KUKA KRL program: EPS_2_25694_BP01_A_20251117072354.src

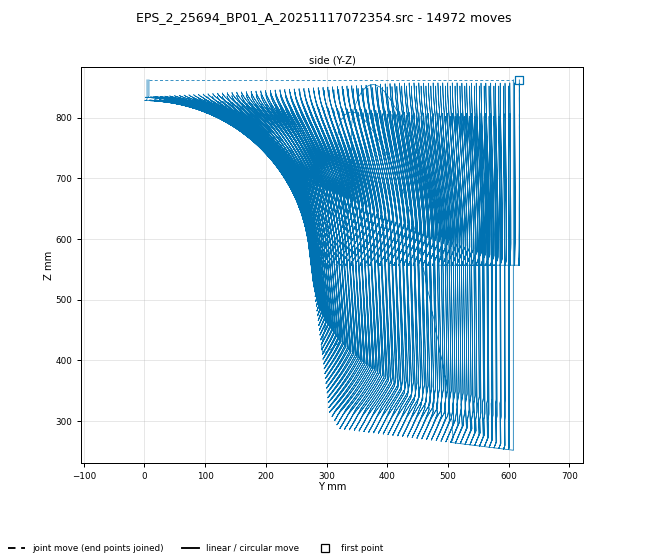
[picture p0: tool path of EPS_2_25694_BP01_A_20251117072354.src, 14972 of 14974 moves have a stored position in this frame; points joined in program order, loops and branches not executed]
&ACCESS RVP
&REL 4
&COMMENT QRS 19112012
&PARAM EDITMASK = *
DEF PART()
EXT BAS (BAS_COMMAND :IN,REAL :IN )
INT I
BAS (#INITMOV,0 )

;KUKA QRS Post kuka4.cps  Date:22-06-2017 !

File_ID=2910

QRS_PRE_INIT()

;Init var - Until changes are made in qrs_pre_init
Outlet_Square_prg=0
Inlet_1_Square_prg=0
Inlet_2_Square_prg=0
Inlet_3_Square_prg=0
Inlet_4_Square_prg=0
Inlet_5_Square_prg=0

Outlet_1={X 0.000, Y 425.000, Z 586.000, B 0.000, E1 0.000 }
Inlet_1={X 0.000, Y 466.000, Z 574.000, B 0.000, E1 180.000 }
Outlet_1_type=533
Inlet_1_type=457
;QRS#1=Sidecore dimensions
;QRS#2=525-21" Concrete
;QRS#3=450-18" Concrete
;QRS#4=
;QRS#5=
;QRS#6=
;QRS#7=
;QRS#8=
;QRS#9=S306-32
;QRS#10=28A PSX-2
;QRS#11=
;QRS#12=
;QRS#13=
;QRS#14=
;QRS#15=
;QRS#16=1220x127x1219 4'
;QRS#17=EPS Height
;QRS#18=852,5
;QRS#19=*
;QRS#20= UPDATED VERSION 22-06-2017
;QRS#21=*
Outlet_Square=0250
Inlet_1_Square=0250
Inlet_2_Square=0
Inlet_3_Square=0
Inlet_4_Square=0
Inlet_5_Square=0
Mill_Square=1
Outlet_Square_Prg=263
Inlet_1_Square_prg=274

QRS_INIT()

$ADVANCE=5

; T1
PTP {E1 171.043,E2 171.043}
PTP {X 0,Y 617.776,A -85,B 0,C 180,E1 171.043,E2 171.043,E3 0,E4 0,E5 0,E6 0}
QRS_SPEED_INIT()
LIN {X 0,Y 617.776,Z 862.5,A -85,B 0,C 180,E1 171.043,E2 171.043,E3 0,E4 0,E5 0,E6 0} C_VEL
LIN {X 0,Y 617.776,Z 559.03,A -85,B 0,C 180,E1 171.043,E2 171.043} C_VEL
LIN {X 0,Y 617.813,Z 557.03,A -85,B 0,C 180,E1 171.228,E2 171.228} C_VEL
LIN {X 0,Y 617.994,Z 557.03,A -85,B 0,C 180,E1 171.886,E2 171.886} C_VEL
LIN {X 0,Y 618.06,Z 557.03,A -85,B 0,C 180,E1 176.532,E2 176.532} C_VEL
LIN {X 0,Y 618.033,Z 557.03,A -85,B 0,C 180,E1 181.155,E2 181.155} C_VEL
LIN {X 0,Y 617.978,Z 557.03,A -85,B 0,C 180,E1 185.787,E2 185.787} C_VEL
LIN {X 0,Y 617.994,Z 557.03,A -85,B 0,C 180,E1 190.456,E2 190.456} C_VEL
LIN {X 0,Y 617.919,Z 557.03,A -85,B 0,C 180,E1 195.199,E2 195.199} C_VEL
LIN {X 0,Y 617.921,Z 557.03,A -85,B 0,C 180,E1 200.05,E2 200.05} C_VEL
LIN {X 0,Y 617.439,Z 557.03,A -85,B 0,C 180,E1 202.548,E2 202.548} C_VEL
LIN {X 0,Y 617.89,Z 557.03,A -85,B 0,C 180,E1 205.057,E2 205.057} C_VEL
LIN {X 0,Y 617.413,Z 557.03,A -85,B 0,C 180,E1 207.659,E2 207.659} C_VEL
LIN {X 0,Y 617.896,Z 557.03,A -85,B 0,C 180,E1 210.277,E2 210.277} C_VEL
LIN {X 0,Y 617.343,Z 557.03,A -85,B 0,C 180,E1 213.025,E2 213.025} C_VEL
LIN {X 0,Y 617.808,Z 557.03,A -85,B 0,C 180,E1 215.799,E2 215.799} C_VEL
LIN {X 0,Y 617.581,Z 557.03,A -85,B 0,C 180,E1 218.103,E2 218.103} C_VEL
LIN {X 0,Y 617.561,Z 557.03,A -85,B 0,C 180,E1 218.721,E2 218.721} C_VEL
LIN {X 0,Y 617.791,Z 557.03,A -85,B 0,C 180,E1 221.731,E2 221.731} C_VEL
LIN {X 0,Y 617.868,Z 557.03,A -85,B 0,C 180,E1 225.1,E2 225.1} C_VEL
LIN {X 0,Y 617.445,Z 557.03,A -85,B 0,C 180,E1 228.309,E2 228.309} C_VEL
LIN {X 0,Y 617.791,Z 557.03,A -85,B 0,C 180,E1 231.298,E2 231.298} C_VEL
LIN {X 0,Y 617.736,Z 557.03,A -85,B 0,C 180,E1 235.8,E2 235.8} C_VEL
LIN {X 0,Y 617.923,Z 557.03,A -85,B 0,C 180,E1 237.011,E2 237.011} C_VEL
LIN {X 0,Y 618.028,Z 557.03,A -85,B 0,C 180,E1 240.51,E2 240.51} C_VEL
LIN {X 0,Y 617.97,Z 557.03,A -85,B 0,C 180,E1 240.75,E2 240.75} C_VEL
LIN {X 0,Y 616.889,Z 557.03,A -85,B 0,C 180,E1 240.936,E2 240.936} C_VEL
LIN {X 0,Y 616.577,Z 557.502,A -85,B 0,C 180,E1 240.975,E2 240.975} C_VEL
LIN {X 0,Y 617.559,Z 570.177,A -85,B 0,C 180,E1 241.191,E2 241.191} C_VEL
LIN {X 0,Y 617.762,Z 600.266,A -85,B 0,C 180,E1 241.598,E2 241.598} C_VEL
LIN {X 0,Y 617.686,Z 612.976,A -85,B 0,C 180,E1 241.802,E2 241.802} C_VEL
LIN {X 0,Y 617.749,Z 625.832,A -85,B 0,C 180,E1 242.076,E2 242.076} C_VEL
LIN {X 0,Y 617.694,Z 639.689,A -85,B 0,C 180,E1 242.437,E2 242.437} C_VEL
LIN {X 0,Y 617.798,Z 652.671,A -85,B 0,C 180,E1 242.849,E2 242.849} C_VEL
LIN {X 0,Y 617.803,Z 663.961,A -85,B 0,C 180,E1 243.254,E2 243.254} C_VEL
LIN {X 0,Y 617.861,Z 675.827,A -85,B 0,C 180,E1 243.741,E2 243.741} C_VEL
LIN {X 0,Y 617.923,Z 689.601,A -85,B 0,C 180,E1 244.386,E2 244.386} C_VEL
LIN {X 0,Y 617.876,Z 701.688,A -85,B 0,C 180,E1 245.016,E2 245.016} C_VEL
LIN {X 0,Y 617.897,Z 713.952,A -85,B 0,C 180,E1 245.732,E2 245.732} C_VEL
LIN {X 0,Y 617.922,Z 724.145,A -85,B 0,C 180,E1 246.381,E2 246.381} C_VEL
LIN {X 0,Y 617.934,Z 735.43,A -85,B 0,C 180,E1 247.172,E2 247.172} C_VEL
LIN {X 0,Y 617.917,Z 745.514,A -85,B 0,C 180,E1 247.939,E2 247.939} C_VEL
LIN {X 0,Y 617.886,Z 756.654,A -85,B 0,C 180,E1 248.87,E2 248.87} C_VEL
LIN {X 0,Y 617.923,Z 766.773,A -85,B 0,C 180,E1 249.797,E2 249.797} C_VEL
LIN {X 0,Y 617.933,Z 775.518,A -85,B 0,C 180,E1 250.667,E2 250.667} C_VEL
LIN {X 0,Y 617.881,Z 782.638,A -85,B 0,C 180,E1 251.422,E2 251.422} C_VEL
LIN {X 0,Y 617.901,Z 791.021,A -85,B 0,C 180,E1 252.392,E2 252.392} C_VEL
LIN {X 0,Y 617.982,Z 799.193,A -85,B 0,C 180,E1 253.428,E2 253.428} C_VEL
LIN {X 0,Y 617.836,Z 807.711,A -85,B 0,C 180,E1 254.61,E2 254.61} C_VEL
LIN {X 0,Y 617.888,Z 814.772,A -85,B 0,C 180,E1 255.697,E2 255.697} C_VEL
LIN {X 0,Y 617.959,Z 820.124,A -85,B 0,C 180,E1 256.591,E2 256.591} C_VEL
LIN {X 0,Y 617.783,Z 826.565,A -85,B 0,C 180,E1 257.773,E2 257.773} C_VEL
LIN {X 0,Y 617.807,Z 832.247,A -85,B 0,C 180,E1 258.953,E2 258.953} C_VEL
LIN {X 0,Y 617.977,Z 836.456,A -85,B 0,C 180,E1 259.949,E2 259.949} C_VEL
LIN {X 0,Y 617.803,Z 841.446,A -85,B 0,C 180,E1 261.247,E2 261.247} C_VEL
LIN {X 0,Y 617.803,Z 845.018,A -85,B 0,C 180,E1 262.35,E2 262.35} C_VEL
LIN {X 0,Y 617.953,Z 848.842,A -85,B 0,C 180,E1 263.749,E2 263.749} C_VEL
LIN {X 0,Y 617.736,Z 851.904,A -85,B 0,C 180,E1 265.14,E2 265.14} C_VEL
LIN {X 0,Y 617.832,Z 854.096,A -85,B 0,C 180,E1 266.531,E2 266.531} C_VEL
LIN {X 0,Y 617.988,Z 855.163,A -85,B 0,C 180,E1 267.458,E2 267.458} C_VEL
LIN {X 0,Y 617.747,Z 856.216,A -85,B 0,C 180,E1 268.844,E2 268.844} C_VEL
LIN {X 0,Y 617.992,Z 856.149,A -85,B 0,C 180,E1 271.155,E2 271.155} C_VEL
LIN {X 0,Y 617.755,Z 855.226,A -85,B 0,C 180,E1 272.543,E2 272.543} C_VEL
LIN {X 0,Y 617.755,Z 854.116,A -85,B 0,C 180,E1 273.469,E2 273.469} C_VEL
LIN {X 0,Y 617.985,Z 851.839,A -85,B 0,C 180,E1 274.858,E2 274.858} C_VEL
LIN {X 0,Y 617.799,Z 848.881,A -85,B 0,C 180,E1 276.253,E2 276.253} C_VEL
LIN {X 0,Y 617.848,Z 845.007,A -85,B 0,C 180,E1 277.649,E2 277.649} C_VEL
LIN {X 0,Y 617.932,Z 841.117,A -85,B 0,C 180,E1 278.831,E2 278.831} C_VEL
LIN {X 0,Y 617.775,Z 836.414,A -85,B 0,C 180,E1 280.075,E2 280.075} C_VEL
LIN {X 0,Y 617.825,Z 832.243,A -85,B 0,C 180,E1 281.047,E2 281.047} C_VEL
LIN {X 0,Y 617.969,Z 826.527,A -85,B 0,C 180,E1 282.224,E2 282.224} C_VEL
LIN {X 0,Y 617.83,Z 820.149,A -85,B 0,C 180,E1 283.411,E2 283.411} C_VEL
LIN {X 0,Y 617.902,Z 811.935,A -85,B 0,C 180,E1 284.75,E2 284.75} C_VEL
LIN {X 0,Y 617.938,Z 805.132,A -85,B 0,C 180,E1 285.758,E2 285.758} C_VEL
LIN {X 0,Y 617.865,Z 798.318,A -85,B 0,C 180,E1 286.693,E2 286.693} C_VEL
LIN {X 0,Y 617.91,Z 789.904,A -85,B 0,C 180,E1 287.74,E2 287.74} C_VEL
LIN {X 0,Y 617.968,Z 781.813,A -85,B 0,C 180,E1 288.665,E2 288.665} C_VEL
LIN {X 0,Y 617.898,Z 771.905,A -85,B 0,C 180,E1 289.703,E2 289.703} C_VEL
LIN {X 0,Y 617.915,Z 763.533,A -85,B 0,C 180,E1 290.511,E2 290.511} C_VEL
LIN {X 0,Y 617.932,Z 753.036,A -85,B 0,C 180,E1 291.438,E2 291.438} C_VEL
LIN {X 0,Y 617.906,Z 743.499,A -85,B 0,C 180,E1 292.217,E2 292.217} C_VEL
LIN {X 0,Y 617.904,Z 733.654,A -85,B 0,C 180,E1 292.959,E2 292.959} C_VEL
LIN {X 0,Y 617.855,Z 722.087,A -85,B 0,C 180,E1 293.756,E2 293.756} C_VEL
LIN {X 0,Y 617.9,Z 709.883,A -85,B 0,C 180,E1 294.513,E2 294.513} C_VEL
LIN {X 0,Y 617.869,Z 698.891,A -85,B 0,C 180,E1 295.137,E2 295.137} C_VEL
LIN {X 0,Y 617.811,Z 688.028,A -85,B 0,C 180,E1 295.699,E2 295.699} C_VEL
LIN {X 0,Y 617.891,Z 673.877,A -85,B 0,C 180,E1 296.338,E2 296.338} C_VEL
LIN {X 0,Y 617.852,Z 660.675,A -85,B 0,C 180,E1 296.865,E2 296.865} C_VEL
LIN {X 0,Y 617.731,Z 650.373,A -85,B 0,C 180,E1 297.236,E2 297.236} C_VEL
LIN {X 0,Y 617.857,Z 634.521,A -85,B 0,C 180,E1 297.699,E2 297.699} C_VEL
LIN {X 0,Y 617.754,Z 621.706,A -85,B 0,C 180,E1 298.018,E2 298.018} C_VEL
LIN {X 0,Y 617.687,Z 613.02,A -85,B 0,C 180,E1 298.197,E2 298.197} C_VEL
LIN {X 0,Y 617.736,Z 606.549,A -85,B 0,C 180,E1 298.307,E2 298.307} C_VEL
LIN {X 0,Y 617.744,Z 594.08,A -85,B 0,C 180,E1 298.49,E2 298.49} C_VEL
LIN {X 0,Y 617.654,Z 580.796,A -85,B 0,C 180,E1 298.667,E2 298.667} C_VEL
LIN {X 0,Y 617.292,Z 566.02,A -85,B 0,C 180,E1 298.877,E2 298.877} C_VEL
LIN {X 0,Y 616.884,Z 557.03,A -85,B 0,C 180,E1 299.063,E2 299.063} C_VEL
LIN {X 0,Y 617.909,Z 557.03,A -85,B 0,C 180,E1 299.23,E2 299.23} C_VEL
LIN {X 0,Y 618.035,Z 557.03,A -85,B 0,C 180,E1 299.444,E2 299.444} C_VEL
LIN {X 0,Y 617.919,Z 557.03,A -85,B 0,C 180,E1 302.989,E2 302.989} C_VEL
LIN {X 0,Y 617.722,Z 557.03,A -85,B 0,C 180,E1 304.198,E2 304.198} C_VEL
LIN {X 0,Y 617.789,Z 557.03,A -85,B 0,C 180,E1 308.703,E2 308.703} C_VEL
LIN {X 0,Y 617.443,Z 557.03,A -85,B 0,C 180,E1 311.758,E2 311.758} C_VEL
LIN {X 0,Y 617.868,Z 557.03,A -85,B 0,C 180,E1 314.9,E2 314.9} C_VEL
LIN {X 0,Y 617.791,Z 557.03,A -85,B 0,C 180,E1 318.271,E2 318.271} C_VEL
LIN {X 0,Y 617.554,Z 557.03,A -85,B 0,C 180,E1 321.278,E2 321.278} C_VEL
LIN {X 0,Y 617.58,Z 557.03,A -85,B 0,C 180,E1 321.897,E2 321.897} C_VEL
LIN {X 0,Y 617.801,Z 557.03,A -85,B 0,C 180,E1 324.201,E2 324.201} C_VEL
LIN {X 0,Y 617.345,Z 557.03,A -85,B 0,C 180,E1 326.975,E2 326.975} C_VEL
LIN {X 0,Y 617.887,Z 557.03,A -85,B 0,C 180,E1 329.722,E2 329.722} C_VEL
LIN {X 0,Y 617.405,Z 557.03,A -85,B 0,C 180,E1 332.34,E2 332.34} C_VEL
LIN {X 0,Y 617.882,Z 557.03,A -85,B 0,C 180,E1 334.943,E2 334.943} C_VEL
LIN {X 0,Y 617.431,Z 557.03,A -85,B 0,C 180,E1 337.451,E2 337.451} C_VEL
LIN {X 0,Y 617.935,Z 557.03,A -85,B 0,C 180,E1 339.951,E2 339.951} C_VEL
LIN {X 0,Y 618,Z 557.03,A -85,B 0,C 180,E1 343.636,E2 343.636} C_VEL
LIN {X 0,Y 617.991,Z 557.03,A -85,B 0,C 180,E1 349.544,E2 349.544} C_VEL
LIN {X 0,Y 617.989,Z 557.03,A -85,B 0,C 180,E1 354.213,E2 354.213} C_VEL
LIN {X 0,Y 618.039,Z 557.03,A -85,B 0,C 180,E1 358.845,E2 358.845} C_VEL
LIN {X 0,Y 618.057,Z 557.03,A -85,B 0,C 180,E1 363.468,E2 363.468} C_VEL
LIN {X 0,Y 618.001,Z 557.03,A -85,B 0,C 180,E1 368.114,E2 368.114} C_VEL
LIN {X 0,Y 617.989,Z 557.03,A -85,B 0,C 180,E1 372.815,E2 372.815} C_VEL
LIN {X 0,Y 617.976,Z 557.03,A -85,B 0,C 180,E1 377.606,E2 377.606} C_VEL
LIN {X 0,Y 617.778,Z 557.03,A -85,B 0,C 180,E1 378.555,E2 378.555} C_VEL
LIN {X 0,Y 617.925,Z 557.03,A -85,B 0,C 180,E1 382.53,E2 382.53} C_VEL
LIN {X 0,Y 617.433,Z 557.03,A -85,B 0,C 180,E1 385.077,E2 385.077} C_VEL
LIN {X 0,Y 617.885,Z 557.03,A -85,B 0,C 180,E1 387.636,E2 387.636} C_VEL
LIN {X 0,Y 617.381,Z 557.03,A -85,B 0,C 180,E1 390.305,E2 390.305} C_VEL
LIN {X 0,Y 617.86,Z 557.03,A -85,B 0,C 180,E1 392.994,E2 392.994} C_VEL
LIN {X 0,Y 617.716,Z 557.03,A -85,B 0,C 180,E1 394.2,E2 394.2} C_VEL
LIN {X 0,Y 617.789,Z 557.03,A -85,B 0,C 180,E1 398.704,E2 398.704} C_VEL
LIN {X 0,Y 617.442,Z 557.03,A -85,B 0,C 180,E1 401.76,E2 401.76} C_VEL
LIN {X 0,Y 617.873,Z 557.03,A -85,B 0,C 180,E1 404.901,E2 404.901} C_VEL
LIN {X 0,Y 617.781,Z 557.03,A -85,B 0,C 180,E1 408.274,E2 408.274} C_VEL
LIN {X 0,Y 617.558,Z 557.03,A -85,B 0,C 180,E1 411.28,E2 411.28} C_VEL
LIN {X 0,Y 617.581,Z 557.03,A -85,B 0,C 180,E1 411.9,E2 411.9} C_VEL
LIN {X 0,Y 617.818,Z 557.03,A -85,B 0,C 180,E1 414.203,E2 414.203} C_VEL
LIN {X 0,Y 617.358,Z 557.03,A -85,B 0,C 180,E1 416.977,E2 416.977} C_VEL
LIN {X 0,Y 617.888,Z 557.03,A -85,B 0,C 180,E1 419.723,E2 419.723} C_VEL
LIN {X 0,Y 618.069,Z 557.03,A -85,B 0,C 180,E1 424.952,E2 424.952} C_VEL
LIN {X 0,Y 617.631,Z 557.03,A -85,B 0,C 180,E1 425.111,E2 425.111} C_VEL
LIN {X 0,Y 617.885,Z 586.594,A -85,B 0,C 180,E1 425.51,E2 425.51} C_VEL
LIN {X 0,Y 617.875,Z 595.62,A -85,B 0,C 180,E1 425.66,E2 425.66} C_VEL
LIN {X 0,Y 617.768,Z 605.441,A -85,B 0,C 180,E1 425.857,E2 425.857} C_VEL
LIN {X 0,Y 617.884,Z 617.86,A -85,B 0,C 180,E1 426.178,E2 426.178} C_VEL
LIN {X 0,Y 617.826,Z 629.53,A -85,B 0,C 180,E1 426.533,E2 426.533} C_VEL
LIN {X 0,Y 617.909,Z 640.015,A -85,B 0,C 180,E1 426.907,E2 426.907} C_VEL
LIN {X 0,Y 617.952,Z 650.109,A -85,B 0,C 180,E1 427.314,E2 427.314} C_VEL
LIN {X 0,Y 617.88,Z 662.072,A -85,B 0,C 180,E1 427.86,E2 427.86} C_VEL
LIN {X 0,Y 617.951,Z 672.651,A -85,B 0,C 180,E1 428.407,E2 428.407} C_VEL
LIN {X 0,Y 617.961,Z 683.449,A -85,B 0,C 180,E1 429.027,E2 429.027} C_VEL
LIN {X 0,Y 617.946,Z 693.19,A -85,B 0,C 180,E1 429.644,E2 429.644} C_VEL
LIN {X 0,Y 617.955,Z 702.637,A -85,B 0,C 180,E1 430.302,E2 430.302} C_VEL
LIN {X 0,Y 617.948,Z 711.779,A -85,B 0,C 180,E1 430.999,E2 430.999} C_VEL
LIN {X 0,Y 617.962,Z 720.66,A -85,B 0,C 180,E1 431.74,E2 431.74} C_VEL
LIN {X 0,Y 617.938,Z 727.924,A -85,B 0,C 180,E1 432.393,E2 432.393} C_VEL
LIN {X 0,Y 617.896,Z 736.057,A -85,B 0,C 180,E1 433.19,E2 433.19} C_VEL
LIN {X 0,Y 617.935,Z 744.033,A -85,B 0,C 180,E1 434.047,E2 434.047} C_VEL
LIN {X 0,Y 617.972,Z 750.526,A -85,B 0,C 180,E1 434.803,E2 434.803} C_VEL
LIN {X 0,Y 617.878,Z 757.608,A -85,B 0,C 180,E1 435.697,E2 435.697} C_VEL
LIN {X 0,Y 617.881,Z 764.039,A -85,B 0,C 180,E1 436.59,E2 436.59} C_VEL
LIN {X 0,Y 617.968,Z 769.873,A -85,B 0,C 180,E1 437.481,E2 437.481} C_VEL
LIN {X 0,Y 617.895,Z 775.211,A -85,B 0,C 180,E1 438.365,E2 438.365} C_VEL
LIN {X 0,Y 617.822,Z 780.028,A -85,B 0,C 180,E1 439.248,E2 439.248} C_VEL
LIN {X 0,Y 617.909,Z 785.055,A -85,B 0,C 180,E1 440.282,E2 440.282} C_VEL
LIN {X 0,Y 617.934,Z 789.878,A -85,B 0,C 180,E1 441.409,E2 441.409} C_VEL
LIN {X 0,Y 617.828,Z 793.427,A -85,B 0,C 180,E1 442.35,E2 442.35} C_VEL
LIN {X 0,Y 617.869,Z 796.435,A -85,B 0,C 180,E1 443.283,E2 443.283} C_VEL
LIN {X 0,Y 617.984,Z 799.004,A -85,B 0,C 180,E1 444.214,E2 444.214} C_VEL
LIN {X 0,Y 617.828,Z 801.242,A -85,B 0,C 180,E1 445.141,E2 445.141} C_VEL
LIN {X 0,Y 617.788,Z 802.267,A -85,B 0,C 180,E1 445.604,E2 445.604} C_VEL
LIN {X 0,Y 617.816,Z 803.833,A -85,B 0,C 180,E1 446.531,E2 446.531} C_VEL
LIN {X 0,Y 617.944,Z 804.995,A -85,B 0,C 180,E1 447.457,E2 447.457} C_VEL
LIN {X 0,Y 617.81,Z 806.19,A -85,B 0,C 180,E1 448.844,E2 448.844} C_VEL
LIN {X 0,Y 617.824,Z 806.4,A -85,B 0,C 180,E1 450.231,E2 450.231} C_VEL
LIN {X 0,Y 617.987,Z 806.076,A -85,B 0,C 180,E1 451.155,E2 451.155} C_VEL
LIN {X 0,Y 617.789,Z 804.929,A -85,B 0,C 180,E1 452.543,E2 452.543} C_VEL
LIN {X 0,Y 617.805,Z 803.683,A -85,B 0,C 180,E1 453.469,E2 453.469} C_VEL
LIN {X 0,Y 617.86,Z 802.891,A -85,B 0,C 180,E1 453.932,E2 453.932} C_VEL
LIN {X 0,Y 617.956,Z 801.012,A -85,B 0,C 180,E1 454.858,E2 454.858} C_VEL
LIN {X 0,Y 617.905,Z 800.019,A -85,B 0,C 180,E1 455.323,E2 455.323} C_VEL
LIN {X 0,Y 617.829,Z 797.557,A -85,B 0,C 180,E1 456.253,E2 456.253} C_VEL
LIN {X 0,Y 617.961,Z 793.056,A -85,B 0,C 180,E1 457.648,E2 457.648} C_VEL
LIN {X 0,Y 617.925,Z 789.897,A -85,B 0,C 180,E1 458.496,E2 458.496} C_VEL
LIN {X 0,Y 617.822,Z 784.889,A -85,B 0,C 180,E1 459.668,E2 459.668} C_VEL
LIN {X 0,Y 617.922,Z 779.516,A -85,B 0,C 180,E1 460.751,E2 460.751} C_VEL
LIN {X 0,Y 617.93,Z 774.69,A -85,B 0,C 180,E1 461.634,E2 461.634} C_VEL
LIN {X 0,Y 617.862,Z 769.352,A -85,B 0,C 180,E1 462.521,E2 462.521} C_VEL
LIN {X 0,Y 617.938,Z 761.307,A -85,B 0,C 180,E1 463.706,E2 463.706} C_VEL
LIN {X 0,Y 617.955,Z 754.609,A -85,B 0,C 180,E1 464.599,E2 464.599} C_VEL
LIN {X 0,Y 617.885,Z 748.243,A -85,B 0,C 180,E1 465.385,E2 465.385} C_VEL
LIN {X 0,Y 617.919,Z 739.516,A -85,B 0,C 180,E1 466.357,E2 466.357} C_VEL
LIN {X 0,Y 617.964,Z 732.409,A -85,B 0,C 180,E1 467.084,E2 467.084} C_VEL
LIN {X 0,Y 617.932,Z 724.143,A -85,B 0,C 180,E1 467.863,E2 467.863} C_VEL
LIN {X 0,Y 617.929,Z 715.725,A -85,B 0,C 180,E1 468.591,E2 468.591} C_VEL
LIN {X 0,Y 617.958,Z 707.441,A -85,B 0,C 180,E1 469.25,E2 469.25} C_VEL
LIN {X 0,Y 617.954,Z 697.702,A -85,B 0,C 180,E1 469.959,E2 469.959} C_VEL
LIN {X 0,Y 617.95,Z 688.245,A -85,B 0,C 180,E1 470.587,E2 470.587} C_VEL
LIN {X 0,Y 617.917,Z 677.977,A -85,B 0,C 180,E1 471.206,E2 471.206} C_VEL
LIN {X 0,Y 617.939,Z 668.024,A -85,B 0,C 180,E1 471.749,E2 471.749} C_VEL
LIN {X 0,Y 617.951,Z 658.602,A -85,B 0,C 180,E1 472.216,E2 472.216} C_VEL
LIN {X 0,Y 617.925,Z 646.97,A -85,B 0,C 180,E1 472.727,E2 472.727} C_VEL
LIN {X 0,Y 617.805,Z 635.606,A -85,B 0,C 180,E1 473.169,E2 473.169} C_VEL
LIN {X 0,Y 617.942,Z 623.528,A -85,B 0,C 180,E1 473.563,E2 473.563} C_VEL
LIN {X 0,Y 617.937,Z 612.732,A -85,B 0,C 180,E1 473.868,E2 473.868} C_VEL
LIN {X 0,Y 617.781,Z 601.296,A -85,B 0,C 180,E1 474.142,E2 474.142} C_VEL
LIN {X 0,Y 617.866,Z 589.784,A -85,B 0,C 180,E1 474.353,E2 474.353} C_VEL
LIN {X 0,Y 617.796,Z 572.713,A -85,B 0,C 180,E1 474.591,E2 474.591} C_VEL
LIN {X 0,Y 617.585,Z 562.233,A -85,B 0,C 180,E1 474.731,E2 474.731} C_VEL
LIN {X 0,Y 617.212,Z 557.03,A -85,B 0,C 180,E1 474.82,E2 474.82} C_VEL
LIN {X 0,Y 617.803,Z 557.03,A -85,B 0,C 180,E1 474.915,E2 474.915} C_VEL
LIN {X 0,Y 618.084,Z 557.03,A -85,B 0,C 180,E1 475.048,E2 475.048} C_VEL
LIN {X 0,Y 617.966,Z 557.03,A -85,B 0,C 180,E1 477.631,E2 477.631} C_VEL
LIN {X 0,Y 617.381,Z 557.03,A -85,B 0,C 180,E1 480.304,E2 480.304} C_VEL
LIN {X 0,Y 617.856,Z 557.03,A -85,B 0,C 180,E1 482.993,E2 482.993} C_VEL
LIN {X 0,Y 617.724,Z 557.03,A -85,B 0,C 180,E1 484.199,E2 484.199} C_VEL
LIN {X 0,Y 617.786,Z 557.03,A -85,B 0,C 180,E1 488.703,E2 488.703} C_VEL
LIN {X 0,Y 617.447,Z 557.03,A -85,B 0,C 180,E1 491.758,E2 491.758} C_VEL
LIN {X 0,Y 617.883,Z 557.03,A -85,B 0,C 180,E1 494.898,E2 494.898} C_VEL
LIN {X 0,Y 617.779,Z 557.03,A -85,B 0,C 180,E1 498.272,E2 498.272} C_VEL
LIN {X 0,Y 617.556,Z 557.03,A -85,B 0,C 180,E1 501.279,E2 501.279} C_VEL
LIN {X 0,Y 617.824,Z 557.03,A -85,B 0,C 180,E1 504.202,E2 504.202} C_VEL
LIN {X 0,Y 617.334,Z 557.03,A -85,B 0,C 180,E1 506.974,E2 506.974} C_VEL
LIN {X 0,Y 617.87,Z 557.03,A -85,B 0,C 180,E1 509.721,E2 509.721} C_VEL
LIN {X 0,Y 617.429,Z 557.03,A -85,B 0,C 180,E1 512.341,E2 512.341} C_VEL
LIN {X 0,Y 617.941,Z 557.03,A -85,B 0,C 180,E1 514.945,E2 514.945} C_VEL
LIN {X 0,Y 617.472,Z 557.03,A -85,B 0,C 180,E1 517.453,E2 517.453} C_VEL
LIN {X 0,Y 617.96,Z 557.03,A -85,B 0,C 180,E1 519.952,E2 519.952} C_VEL
LIN {X 0,Y 617.719,Z 557.03,A -85,B 0,C 180,E1 522.386,E2 522.386} C_VEL
LIN {X 0,Y 617.802,Z 557.03,A -85,B 0,C 180,E1 524.798,E2 524.798} C_VEL
LIN {X 0,Y 617.989,Z 557.03,A -85,B 0,C 180,E1 527.185,E2 527.185} C_VEL
LIN {X 0,Y 617.813,Z 557.03,A -85,B 0,C 180,E1 531.228,E2 531.228} C_VEL
LIN {X 0,Y 615.296,Z 557.03,A -85,B 0,C 180,E1 532.425,E2 532.425} C_VEL
LIN {X 0,Y 609.724,Z 557.03,A -85,B 0,C 180,E1 534.213,E2 534.213} C_VEL
LIN {X 0,Y 609.639,Z 557.03,A -85,B 0,C 180,E1 534.42,E2 534.42} C_VEL
LIN {X 0,Y 609.652,Z 557.03,A -85,B 0,C 180,E1 538.577,E2 538.577} C_VEL
LIN {X 0,Y 609.657,Z 557.03,A -85,B 0,C 180,E1 542.847,E2 542.847} C_VEL
LIN {X 0,Y 609.692,Z 557.03,A -85,B 0,C 180,E1 547.132,E2 547.132} C_VEL
LIN {X 0,Y 609.751,Z 557.03,A -85,B 0,C 180,E1 551.457,E2 551.457} C_VEL
LIN {X 0,Y 609.759,Z 557.03,A -85,B 0,C 180,E1 555.85,E2 555.85} C_VEL
LIN {X 0,Y 609.931,Z 557.03,A -85,B 0,C 180,E1 560.335,E2 560.335} C_VEL
LIN {X 0,Y 609.974,Z 557.03,A -85,B 0,C 180,E1 564.957,E2 564.957} C_VEL
LIN {X 0,Y 609.807,Z 557.03,A -85,B 0,C 180,E1 569.771,E2 569.771} C_VEL
LIN {X 0,Y 609.75,Z 557.03,A -85,B 0,C 180,E1 576.577,E2 576.577} C_VEL
LIN {X 0,Y 609.796,Z 557.03,A -85,B 0,C 180,E1 582.093,E2 582.093} C_VEL
LIN {X 0,Y 609.51,Z 557.03,A -85,B 0,C 180,E1 587.88,E2 587.88} C_VEL
LIN {X 0,Y 609.49,Z 557.03,A -85,B 0,C 180,E1 592.643,E2 592.643} C_VEL
LIN {X 0,Y 609.91,Z 557.03,A -85,B 0,C 180,E1 597.561,E2 597.561} C_VEL
LIN {X 0,Y 609.747,Z 557.03,A -85,B 0,C 180,E1 600.607,E2 600.607} C_VEL
LIN {X 0,Y 610.755,Z 624.717,A -85,B 0,C 180,E1 601.699,E2 601.699} C_VEL
LIN {X 0,Y 610.672,Z 664.778,A -85,B 0,C 180,E1 602.95,E2 602.95} C_VEL
LIN {X 0,Y 610.552,Z 703.016,A -85,B 0,C 180,E1 604.773,E2 604.773} C_VEL
LIN {X 0,Y 610.424,Z 738.38,A -85,B 0,C 180,E1 607.102,E2 607.102} C_VEL
LIN {X 0,Y 610.275,Z 769.485,A -85,B 0,C 180,E1 609.799,E2 609.799} C_VEL
LIN {X 0,Y 610.202,Z 796.701,A -85,B 0,C 180,E1 612.864,E2 612.864} C_VEL
LIN {X 0,Y 610.142,Z 820.255,A -85,B 0,C 180,E1 616.365,E2 616.365} C_VEL
LIN {X 0,Y 610.146,Z 837.909,A -85,B 0,C 180,E1 619.997,E2 619.997} C_VEL
LIN {X 0,Y 610.093,Z 849.345,A -85,B 0,C 180,E1 623.517,E2 623.517} C_VEL
LIN {X 0,Y 610.095,Z 855.895,A -85,B 0,C 180,E1 627.155,E2 627.155} C_VEL
LIN {X 0,Y 609.976,Z 857.5,A -85,B 0,C 180,E1 630,E2 630} C_VEL
LIN {X 0,Y 609.92,Z 855.894,A -85,B 0,C 180,E1 632.846,E2 632.846} C_VEL
LIN {X 0,Y 610.022,Z 851.178,A -85,B 0,C 180,E1 635.698,E2 635.698} C_VEL
LIN {X 0,Y 610.036,Z 840.616,A -85,B 0,C 180,E1 639.284,E2 639.284} C_VEL
LIN {X 0,Y 610.133,Z 826.219,A -85,B 0,C 180,E1 642.541,E2 642.541} C_VEL
LIN {X 0,Y 610.147,Z 804.949,A -85,B 0,C 180,E1 646.026,E2 646.026} C_VEL
LIN {X 0,Y 610.251,Z 778.824,A -85,B 0,C 180,E1 649.237,E2 649.237} C_VEL
LIN {X 0,Y 610.37,Z 749.237,A -85,B 0,C 180,E1 652.036,E2 652.036} C_VEL
LIN {X 0,Y 610.51,Z 715.135,A -85,B 0,C 180,E1 654.506,E2 654.506} C_VEL
LIN {X 0,Y 610.67,Z 678.761,A -85,B 0,C 180,E1 656.456,E2 656.456} C_VEL
LIN {X 0,Y 610.794,Z 641.057,A -85,B 0,C 180,E1 657.859,E2 657.859} C_VEL
LIN {X 0,Y 610.787,Z 603.628,A -85,B 0,C 180,E1 658.704,E2 658.704} C_VEL
LIN {X 0,Y 610.127,Z 557.03,A -85,B 0,C 180,E1 659.45,E2 659.45} C_VEL
LIN {X 0,Y 610.009,Z 557.03,A -85,B 0,C 180,E1 663.096,E2 663.096} C_VEL
LIN {X 0,Y 609.592,Z 557.03,A -85,B 0,C 180,E1 669.655,E2 669.655} C_VEL
LIN {X 0,Y 609.744,Z 557.03,A -85,B 0,C 180,E1 675.955,E2 675.955} C_VEL
LIN {X 0,Y 609.562,Z 557.03,A -85,B 0,C 180,E1 680.353,E2 680.353} C_VEL
LIN {X 0,Y 609.598,Z 557.03,A -85,B 0,C 180,E1 685.165,E2 685.165} C_VEL
LIN {X 0,Y 609.765,Z 557.03,A -85,B 0,C 180,E1 690.349,E2 690.349} C_VEL
LIN {X 0,Y 609.957,Z 557.03,A -85,B 0,C 180,E1 695.042,E2 695.042} C_VEL
LIN {X 0,Y 609.776,Z 557.03,A -85,B 0,C 180,E1 701.17,E2 701.17} C_VEL
LIN {X 0,Y 609.349,Z 557.03,A -85,B 0,C 180,E1 705.705,E2 705.705} C_VEL
LIN {X 0,Y 609.921,Z 557.03,A -85,B 0,C 180,E1 709.994,E2 709.994} C_VEL
LIN {X 0,Y 610.069,Z 557.03,A -85,B 0,C 180,E1 714.303,E2 714.303} C_VEL
LIN {X 0,Y 609.771,Z 557.03,A -85,B 0,C 180,E1 720,E2 720} C_VEL
LIN {X 0,Y 609.862,Z 557.03,A -85,B 0,C 180,E1 724.271,E2 724.271} C_VEL
LIN {X 0,Y 609.932,Z 557.03,A -85,B 0,C 180,E1 728.565,E2 728.565} C_VEL
LIN {X 0,Y 610.043,Z 557.03,A -85,B 0,C 180,E1 732.906,E2 732.906} C_VEL
LIN {X 0,Y 609.797,Z 557.03,A -85,B 0,C 180,E1 738.829,E2 738.829} C_VEL
LIN {X 0,Y 609.745,Z 557.03,A -85,B 0,C 180,E1 743.407,E2 743.407} C_VEL
LIN {X 0,Y 609.792,Z 557.03,A -85,B 0,C 180,E1 748.146,E2 748.146} C_VEL
LIN {X 0,Y 609.936,Z 557.03,A -85,B 0,C 180,E1 753.097,E2 753.097} C_VEL
LIN {X 0,Y 609.593,Z 557.03,A -85,B 0,C 180,E1 759.65,E2 759.65} C_VEL
LIN {X 0,Y 609.743,Z 557.03,A -85,B 0,C 180,E1 765.951,E2 765.951} C_VEL
LIN {X 0,Y 609.546,Z 557.03,A -85,B 0,C 180,E1 770.349,E2 770.349} C_VEL
LIN {X 0,Y 609.614,Z 557.03,A -85,B 0,C 180,E1 775.163,E2 775.163} C_VEL
LIN {X 0,Y 609.74,Z 557.03,A -85,B 0,C 180,E1 780.345,E2 780.345} C_VEL
LIN {X 0,Y 610.09,Z 557.03,A -85,B 0,C 180,E1 784.767,E2 784.767} C_VEL
LIN {X 0,Y 610.565,Z 608.543,A -85,B 0,C 180,E1 785.631,E2 785.631} C_VEL
LIN {X 0,Y 610.588,Z 644.002,A -85,B 0,C 180,E1 786.774,E2 786.774} C_VEL
LIN {X 0,Y 610.493,Z 678.24,A -85,B 0,C 180,E1 788.447,E2 788.447} C_VEL
LIN {X 0,Y 610.33,Z 710.6,A -85,B 0,C 180,E1 790.654,E2 790.654} C_VEL
LIN {X 0,Y 610.182,Z 738.67,A -85,B 0,C 180,E1 793.234,E2 793.234} C_VEL
LIN {X 0,Y 610.117,Z 762.804,A -85,B 0,C 180,E1 796.181,E2 796.181} C_VEL
LIN {X 0,Y 610.024,Z 781.443,A -85,B 0,C 180,E1 799.272,E2 799.272} C_VEL
LIN {X 0,Y 610.035,Z 794.648,A -85,B 0,C 180,E1 802.373,E2 802.373} C_VEL
LIN {X 0,Y 609.953,Z 803.546,A -85,B 0,C 180,E1 805.729,E2 805.729} C_VEL
LIN {X 0,Y 609.982,Z 807.039,A -85,B 0,C 180,E1 808.577,E2 808.577} C_VEL
LIN {X 0,Y 610.101,Z 806.975,A -85,B 0,C 180,E1 811.422,E2 811.422} C_VEL
LIN {X 0,Y 610.116,Z 801.854,A -85,B 0,C 180,E1 814.982,E2 814.982} C_VEL
LIN {X 0,Y 610.11,Z 790.83,A -85,B 0,C 180,E1 818.563,E2 818.563} C_VEL
LIN {X 0,Y 610.097,Z 773.941,A -85,B 0,C 180,E1 821.995,E2 821.995} C_VEL
LIN {X 0,Y 610.179,Z 753.827,A -85,B 0,C 180,E1 824.924,E2 824.924} C_VEL
LIN {X 0,Y 610.275,Z 728.541,A -85,B 0,C 180,E1 827.693,E2 827.693} C_VEL
LIN {X 0,Y 610.393,Z 697.993,A -85,B 0,C 180,E1 830.198,E2 830.198} C_VEL
LIN {X 0,Y 610.51,Z 666.105,A -85,B 0,C 180,E1 832.126,E2 832.126} C_VEL
LIN {X 0,Y 610.587,Z 631.823,A -85,B 0,C 180,E1 833.592,E2 833.592} C_VEL
LIN {X 0,Y 610.622,Z 596.548,A -85,B 0,C 180,E1 834.539,E2 834.539} C_VEL
LIN {X 0,Y 610.134,Z 557.03,A -85,B 0,C 180,E1 835.148,E2 835.148} C_VEL
LIN {X 0,Y 609.5,Z 557.03,A -85,B 0,C 180,E1 839.789,E2 839.789} C_VEL
LIN {X 0,Y 609.933,Z 557.03,A -85,B 0,C 180,E1 843.1,E2 843.1} C_VEL
LIN {X 0,Y 609.606,Z 557.03,A -85,B 0,C 180,E1 849.657,E2 849.657} C_VEL
LIN {X 0,Y 609.728,Z 557.03,A -85,B 0,C 180,E1 855.954,E2 855.954} C_VEL
LIN {X 0,Y 609.545,Z 557.03,A -85,B 0,C 180,E1 860.354,E2 860.354} C_VEL
LIN {X 0,Y 609.604,Z 557.03,A -85,B 0,C 180,E1 865.166,E2 865.166} C_VEL
LIN {X 0,Y 609.752,Z 557.03,A -85,B 0,C 180,E1 870.35,E2 870.35} C_VEL
LIN {X 0,Y 610.023,Z 557.03,A -85,B 0,C 180,E1 875.046,E2 875.046} C_VEL
LIN {X 0,Y 609.829,Z 557.03,A -85,B 0,C 180,E1 881.172,E2 881.172} C_VEL
LIN {X 0,Y 610.076,Z 557.03,A -85,B 0,C 180,E1 887.095,E2 887.095} C_VEL
LIN {X 0,Y 609.787,Z 557.03,A -85,B 0,C 180,E1 892.869,E2 892.869} C_VEL
LIN {X 0,Y 609.639,Z 557.03,A -85,B 0,C 180,E1 894.42,E2 894.42} C_VEL
LIN {X 0,Y 605.885,Z 557.03,A -85,B 0,C 180,E1 896.027,E2 896.027} C_VEL
LIN {X 0,Y 601.88,Z 557.03,A -85,B 0,C 180,E1 897.654,E2 897.654} C_VEL
LIN {X 0,Y 602.127,Z 557.03,A -85,B 0,C 180,E1 901.441,E2 901.441} C_VEL
LIN {X 0,Y 602.133,Z 557.03,A -85,B 0,C 180,E1 905.772,E2 905.772} C_VEL
LIN {X 0,Y 601.827,Z 557.03,A -85,B 0,C 180,E1 911.61,E2 911.61} C_VEL
LIN {X 0,Y 601.792,Z 557.03,A -85,B 0,C 180,E1 916.065,E2 916.065} C_VEL
LIN {X 0,Y 601.726,Z 557.03,A -85,B 0,C 180,E1 921.412,E2 921.412} C_VEL
LIN {X 0,Y 601.955,Z 557.03,A -85,B 0,C 180,E1 925.313,E2 925.313} C_VEL
LIN {X 0,Y 601.716,Z 557.03,A -85,B 0,C 180,E1 931.184,E2 931.184} C_VEL
LIN {X 0,Y 601.774,Z 557.03,A -85,B 0,C 180,E1 937.142,E2 937.142} C_VEL
LIN {X 0,Y 601.771,Z 557.03,A -85,B 0,C 180,E1 943.144,E2 943.144} C_VEL
LIN {X 0,Y 601.573,Z 557.03,A -85,B 0,C 180,E1 949.128,E2 949.128} C_VEL
LIN {X 0,Y 601.504,Z 557.03,A -85,B 0,C 180,E1 953.651,E2 953.651} C_VEL
LIN {X 0,Y 601.946,Z 557.03,A -85,B 0,C 180,E1 958.116,E2 958.116} C_VEL
LIN {X 0,Y 602.141,Z 557.03,A -85,B 0,C 180,E1 960.199,E2 960.199} C_VEL
LIN {X 0,Y 603.848,Z 584.523,A -85,B 0,C 180,E1 960.665,E2 960.665} C_VEL
LIN {X 0,Y 603.743,Z 628.413,A -85,B 0,C 180,E1 961.436,E2 961.436} C_VEL
LIN {X 0,Y 603.548,Z 666.152,A -85,B 0,C 180,E1 962.662,E2 962.662} C_VEL
LIN {X 0,Y 603.25,Z 703.692,A -85,B 0,C 180,E1 964.485,E2 964.485} C_VEL
LIN {X 0,Y 602.941,Z 738.47,A -85,B 0,C 180,E1 966.808,E2 966.808} C_VEL
LIN {X 0,Y 602.66,Z 769.298,A -85,B 0,C 180,E1 969.514,E2 969.514} C_VEL
LIN {X 0,Y 602.43,Z 796.874,A -85,B 0,C 180,E1 972.658,E2 972.658} C_VEL
LIN {X 0,Y 602.287,Z 820.256,A -85,B 0,C 180,E1 976.184,E2 976.184} C_VEL
LIN {X 0,Y 602.248,Z 837.908,A -85,B 0,C 180,E1 979.865,E2 979.865} C_VEL
LIN {X 0,Y 602.18,Z 850.114,A -85,B 0,C 180,E1 983.733,E2 983.733} C_VEL
LIN {X 0,Y 602.186,Z 855.895,A -85,B 0,C 180,E1 987.118,E2 987.118} C_VEL
LIN {X 0,Y 602.076,Z 857.5,A -85,B 0,C 180,E1 990,E2 990} C_VEL
LIN {X 0,Y 602.025,Z 855.894,A -85,B 0,C 180,E1 992.883,E2 992.883} C_VEL
LIN {X 0,Y 602.102,Z 850.195,A -85,B 0,C 180,E1 996.231,E2 996.231} C_VEL
LIN {X 0,Y 602.093,Z 839.273,A -85,B 0,C 180,E1 999.773,E2 999.773} C_VEL
LIN {X 0,Y 602.188,Z 822.288,A -85,B 0,C 180,E1 1003.449,E2 1003.449} C_VEL
LIN {X 0,Y 602.356,Z 799.929,A -85,B 0,C 180,E1 1006.943,E2 1006.943} C_VEL
LIN {X 0,Y 602.617,Z 772.522,A -85,B 0,C 180,E1 1010.165,E2 1010.165} C_VEL
LIN {X 0,Y 602.903,Z 740.835,A -85,B 0,C 180,E1 1013.009,E2 1013.009} C_VEL
LIN {X 0,Y 603.221,Z 707.053,A -85,B 0,C 180,E1 1015.318,E2 1015.318} C_VEL
LIN {X 0,Y 603.558,Z 671.389,A -85,B 0,C 180,E1 1017.118,E2 1017.118} C_VEL
LIN {X 0,Y 603.804,Z 634.026,A -85,B 0,C 180,E1 1018.415,E2 1018.415} C_VEL
LIN {X 0,Y 603.875,Z 593.617,A -85,B 0,C 180,E1 1019.213,E2 1019.213} C_VEL
LIN {X 0,Y 602.534,Z 559.493,A -85,B 0,C 180,E1 1019.742,E2 1019.742} C_VEL
LIN {X 0,Y 602.139,Z 557.03,A -85,B 0,C 180,E1 1019.8,E2 1019.8} C_VEL
LIN {X 0,Y 601.592,Z 557.03,A -85,B 0,C 180,E1 1025.37,E2 1025.37} C_VEL
LIN {X 0,Y 601.756,Z 557.03,A -85,B 0,C 180,E1 1028.978,E2 1028.978} C_VEL
LIN {X 0,Y 601.747,Z 557.03,A -85,B 0,C 180,E1 1035.214,E2 1035.214} C_VEL
LIN {X 0,Y 601.738,Z 557.03,A -85,B 0,C 180,E1 1041.261,E2 1041.261} C_VEL
LIN {X 0,Y 601.537,Z 557.03,A -85,B 0,C 180,E1 1046.379,E2 1046.379} C_VEL
LIN {X 0,Y 601.657,Z 557.03,A -85,B 0,C 180,E1 1051.439,E2 1051.439} C_VEL
LIN {X 0,Y 601.702,Z 557.03,A -85,B 0,C 180,E1 1056.26,E2 1056.26} C_VEL
LIN {X 0,Y 601.925,Z 557.03,A -85,B 0,C 180,E1 1060.915,E2 1060.915} C_VEL
LIN {X 0,Y 601.512,Z 557.03,A -85,B 0,C 180,E1 1065.422,E2 1065.422} C_VEL
LIN {X 0,Y 601.977,Z 557.03,A -85,B 0,C 180,E1 1069.86,E2 1069.86} C_VEL
LIN {X 0,Y 602.159,Z 557.03,A -85,B 0,C 180,E1 1074.228,E2 1074.228} C_VEL
LIN {X 0,Y 601.87,Z 557.03,A -85,B 0,C 180,E1 1080,E2 1080} C_VEL
LIN {X 0,Y 601.974,Z 557.03,A -85,B 0,C 180,E1 1084.327,E2 1084.327} C_VEL
LIN {X 0,Y 601.991,Z 557.03,A -85,B 0,C 180,E1 1088.678,E2 1088.678} C_VEL
LIN {X 0,Y 602.068,Z 557.03,A -85,B 0,C 180,E1 1093.08,E2 1093.08} C_VEL
LIN {X 0,Y 601.852,Z 557.03,A -85,B 0,C 180,E1 1099.087,E2 1099.087} C_VEL
LIN {X 0,Y 601.764,Z 557.03,A -85,B 0,C 180,E1 1103.736,E2 1103.736} C_VEL
LIN {X 0,Y 601.776,Z 557.03,A -85,B 0,C 180,E1 1108.555,E2 1108.555} C_VEL
LIN {X 0,Y 601.826,Z 557.03,A -85,B 0,C 180,E1 1113.88,E2 1113.88} C_VEL
LIN {X 0,Y 601.758,Z 557.03,A -85,B 0,C 180,E1 1118.974,E2 1118.974} C_VEL
LIN {X 0,Y 601.736,Z 557.03,A -85,B 0,C 180,E1 1125.209,E2 1125.209} C_VEL
LIN {X 0,Y 601.701,Z 557.03,A -85,B 0,C 180,E1 1131.018,E2 1131.018} C_VEL
LIN {X 0,Y 601.567,Z 557.03,A -85,B 0,C 180,E1 1136.15,E2 1136.15} C_VEL
LIN {X 0,Y 601.614,Z 557.03,A -85,B 0,C 180,E1 1141.434,E2 1141.434} C_VEL
LIN {X 0,Y 602.044,Z 557.252,A -85,B 0,C 180,E1 1144.43,E2 1144.43} C_VEL
LIN {X 0,Y 603.411,Z 568.824,A -85,B 0,C 180,E1 1144.641,E2 1144.641} C_VEL
LIN {X 0,Y 603.337,Z 609.405,A -85,B 0,C 180,E1 1145.342,E2 1145.342} C_VEL
LIN {X 0,Y 603.262,Z 645.08,A -85,B 0,C 180,E1 1146.52,E2 1146.52} C_VEL
LIN {X 0,Y 603.022,Z 679.976,A -85,B 0,C 180,E1 1148.266,E2 1148.266} C_VEL
LIN {X 0,Y 602.69,Z 712.211,A -85,B 0,C 180,E1 1150.534,E2 1150.534} C_VEL
LIN {X 0,Y 602.436,Z 740.269,A -85,B 0,C 180,E1 1153.184,E2 1153.184} C_VEL
LIN {X 0,Y 602.285,Z 764.077,A -85,B 0,C 180,E1 1156.183,E2 1156.183} C_VEL
LIN {X 0,Y 602.159,Z 782.046,A -85,B 0,C 180,E1 1159.257,E2 1159.257} C_VEL
LIN {X 0,Y 602.137,Z 795.1,A -85,B 0,C 180,E1 1162.414,E2 1162.414} C_VEL
LIN {X 0,Y 602.077,Z 803.545,A -85,B 0,C 180,E1 1165.673,E2 1165.673} C_VEL
LIN {X 0,Y 602.081,Z 807.039,A -85,B 0,C 180,E1 1168.559,E2 1168.559} C_VEL
LIN {X 0,Y 602.196,Z 806.976,A -85,B 0,C 180,E1 1171.44,E2 1171.44} C_VEL
LIN {X 0,Y 602.223,Z 801.856,A -85,B 0,C 180,E1 1175.048,E2 1175.048} C_VEL
LIN {X 0,Y 602.208,Z 790.832,A -85,B 0,C 180,E1 1178.676,E2 1178.676} C_VEL
LIN {X 0,Y 602.248,Z 773.946,A -85,B 0,C 180,E1 1182.154,E2 1182.154} C_VEL
LIN {X 0,Y 602.372,Z 752.412,A -85,B 0,C 180,E1 1185.302,E2 1185.302} C_VEL
LIN {X 0,Y 602.603,Z 725.585,A -85,B 0,C 180,E1 1188.209,E2 1188.209} C_VEL
LIN {X 0,Y 602.842,Z 695.212,A -85,B 0,C 180,E1 1190.657,E2 1190.657} C_VEL
LIN {X 0,Y 603.122,Z 661.637,A -85,B 0,C 180,E1 1192.643,E2 1192.643} C_VEL
LIN {X 0,Y 603.398,Z 625.396,A -85,B 0,C 180,E1 1194.112,E2 1194.112} C_VEL
LIN {X 0,Y 603.517,Z 591.367,A -85,B 0,C 180,E1 1194.949,E2 1194.949} C_VEL
LIN {X 0,Y 602.542,Z 559.327,A -85,B 0,C 180,E1 1195.431,E2 1195.431} C_VEL
LIN {X 0,Y 602.186,Z 557.03,A -85,B 0,C 180,E1 1195.523,E2 1195.523} C_VEL
LIN {X 0,Y 601.609,Z 557.03,A -85,B 0,C 180,E1 1201.174,E2 1201.174} C_VEL
LIN {X 0,Y 601.595,Z 557.03,A -85,B 0,C 180,E1 1205.369,E2 1205.369} C_VEL
LIN {X 0,Y 601.761,Z 557.03,A -85,B 0,C 180,E1 1208.977,E2 1208.977} C_VEL
LIN {X 0,Y 601.737,Z 557.03,A -85,B 0,C 180,E1 1215.214,E2 1215.214} C_VEL
LIN {X 0,Y 601.678,Z 557.03,A -85,B 0,C 180,E1 1221.02,E2 1221.02} C_VEL
LIN {X 0,Y 601.544,Z 557.03,A -85,B 0,C 180,E1 1226.159,E2 1226.159} C_VEL
LIN {X 0,Y 601.654,Z 557.03,A -85,B 0,C 180,E1 1231.439,E2 1231.439} C_VEL
LIN {X 0,Y 601.767,Z 557.03,A -85,B 0,C 180,E1 1236.264,E2 1236.264} C_VEL
LIN {X 0,Y 601.956,Z 557.03,A -85,B 0,C 180,E1 1240.916,E2 1240.916} C_VEL
LIN {X 0,Y 602.129,Z 557.03,A -85,B 0,C 180,E1 1246.922,E2 1246.922} C_VEL
LIN {X 0,Y 601.888,Z 557.03,A -85,B 0,C 180,E1 1252.775,E2 1252.775} C_VEL
LIN {X 0,Y 601.88,Z 557.03,A -85,B 0,C 180,E1 1257.654,E2 1257.654} C_VEL
LIN {X 0,Y 597.816,Z 557.03,A -85,B 0,C 180,E1 1259.279,E2 1259.279} C_VEL
LIN {X 0,Y 594.086,Z 557.03,A -85,B 0,C 180,E1 1260.924,E2 1260.924} C_VEL
LIN {X 0,Y 594.078,Z 557.03,A -85,B 0,C 180,E1 1266.312,E2 1266.312} C_VEL
LIN {X 0,Y 593.89,Z 557.03,A -85,B 0,C 180,E1 1271.767,E2 1271.767} C_VEL
LIN {X 0,Y 593.849,Z 557.03,A -85,B 0,C 180,E1 1276.286,E2 1276.286} C_VEL
LIN {X 0,Y 593.947,Z 557.03,A -85,B 0,C 180,E1 1280.907,E2 1280.907} C_VEL
LIN {X 0,Y 593.938,Z 557.03,A -85,B 0,C 180,E1 1285.679,E2 1285.679} C_VEL
LIN {X 0,Y 593.861,Z 557.03,A -85,B 0,C 180,E1 1290.655,E2 1290.655} C_VEL
LIN {X 0,Y 593.849,Z 557.03,A -85,B 0,C 180,E1 1295.899,E2 1295.899} C_VEL
LIN {X 0,Y 593.803,Z 557.03,A -85,B 0,C 180,E1 1301.521,E2 1301.521} C_VEL
LIN {X 0,Y 593.711,Z 557.03,A -85,B 0,C 180,E1 1306.486,E2 1306.486} C_VEL
LIN {X 0,Y 593.697,Z 557.03,A -85,B 0,C 180,E1 1312.262,E2 1312.262} C_VEL
LIN {X 0,Y 593.991,Z 557.03,A -85,B 0,C 180,E1 1317.638,E2 1317.638} C_VEL
LIN {X 0,Y 594.175,Z 557.689,A -85,B 0,C 180,E1 1319.772,E2 1319.772} C_VEL
LIN {X 0,Y 596.436,Z 566.623,A -85,B 0,C 180,E1 1320.02,E2 1320.02} C_VEL
LIN {X 0,Y 596.837,Z 625.38,A -85,B 0,C 180,E1 1320.995,E2 1320.995} C_VEL
LIN {X 0,Y 596.468,Z 664.754,A -85,B 0,C 180,E1 1322.25,E2 1322.25} C_VEL
LIN {X 0,Y 596.03,Z 702.511,A -85,B 0,C 180,E1 1324.083,E2 1324.083} C_VEL
LIN {X 0,Y 595.5,Z 737.235,A -85,B 0,C 180,E1 1326.403,E2 1326.403} C_VEL
LIN {X 0,Y 595.022,Z 768.24,A -85,B 0,C 180,E1 1329.131,E2 1329.131} C_VEL
LIN {X 0,Y 594.671,Z 795.234,A -85,B 0,C 180,E1 1332.211,E2 1332.211} C_VEL
LIN {X 0,Y 594.462,Z 816.852,A -85,B 0,C 180,E1 1335.413,E2 1335.413} C_VEL
LIN {X 0,Y 594.292,Z 834.674,A -85,B 0,C 180,E1 1338.949,E2 1338.949} C_VEL
LIN {X 0,Y 594.213,Z 847.614,A -85,B 0,C 180,E1 1342.681,E2 1342.681} C_VEL
LIN {X 0,Y 594.154,Z 853.932,A -85,B 0,C 180,E1 1345.616,E2 1345.616} C_VEL
LIN {X 0,Y 594.164,Z 857.083,A -85,B 0,C 180,E1 1348.54,E2 1348.54} C_VEL
LIN {X 0,Y 594.298,Z 857.082,A -85,B 0,C 180,E1 1351.46,E2 1351.46} C_VEL
LIN {X 0,Y 594.393,Z 852.725,A -85,B 0,C 180,E1 1355.115,E2 1355.115} C_VEL
LIN {X 0,Y 594.304,Z 841.96,A -85,B 0,C 180,E1 1359.162,E2 1359.162} C_VEL
LIN {X 0,Y 594.401,Z 826.221,A -85,B 0,C 180,E1 1362.878,E2 1362.878} C_VEL
LIN {X 0,Y 594.569,Z 806.285,A -85,B 0,C 180,E1 1366.267,E2 1366.267} C_VEL
LIN {X 0,Y 594.903,Z 779.517,A -85,B 0,C 180,E1 1369.678,E2 1369.678} C_VEL
LIN {X 0,Y 595.292,Z 749.585,A -85,B 0,C 180,E1 1372.595,E2 1372.595} C_VEL
LIN {X 0,Y 595.806,Z 715.444,A -85,B 0,C 180,E1 1375.132,E2 1375.132} C_VEL
LIN {X 0,Y 596.358,Z 678.814,A -85,B 0,C 180,E1 1377.14,E2 1377.14} C_VEL
LIN {X 0,Y 596.751,Z 641.679,A -85,B 0,C 180,E1 1378.555,E2 1378.555} C_VEL
LIN {X 0,Y 596.97,Z 604.607,A -85,B 0,C 180,E1 1379.417,E2 1379.417} C_VEL
LIN {X 0,Y 595.9,Z 562.031,A -85,B 0,C 180,E1 1380.072,E2 1380.072} C_VEL
LIN {X 0,Y 594.107,Z 557.03,A -85,B 0,C 180,E1 1380.291,E2 1380.291} C_VEL
LIN {X 0,Y 593.629,Z 557.03,A -85,B 0,C 180,E1 1385.917,E2 1385.917} C_VEL
LIN {X 0,Y 593.623,Z 557.03,A -85,B 0,C 180,E1 1391.54,E2 1391.54} C_VEL
LIN {X 0,Y 593.831,Z 557.03,A -85,B 0,C 180,E1 1396.5,E2 1396.5} C_VEL
LIN {X 0,Y 593.818,Z 557.03,A -85,B 0,C 180,E1 1402.274,E2 1402.274} C_VEL
LIN {X 0,Y 593.658,Z 557.03,A -85,B 0,C 180,E1 1407.619,E2 1407.619} C_VEL
LIN {X 0,Y 593.718,Z 557.03,A -85,B 0,C 180,E1 1412.678,E2 1412.678} C_VEL
LIN {X 0,Y 593.705,Z 557.03,A -85,B 0,C 180,E1 1417.511,E2 1417.511} C_VEL
LIN {X 0,Y 593.992,Z 557.03,A -85,B 0,C 180,E1 1422.19,E2 1422.19} C_VEL
LIN {X 0,Y 593.736,Z 557.03,A -85,B 0,C 180,E1 1428.229,E2 1428.229} C_VEL
LIN {X 0,Y 594.223,Z 557.03,A -85,B 0,C 180,E1 1434.151,E2 1434.151} C_VEL
LIN {X 0,Y 593.969,Z 557.03,A -85,B 0,C 180,E1 1440,E2 1440} C_VEL
LIN {X 0,Y 594.057,Z 557.03,A -85,B 0,C 180,E1 1444.385,E2 1444.385} C_VEL
LIN {X 0,Y 594.071,Z 557.03,A -85,B 0,C 180,E1 1448.795,E2 1448.795} C_VEL
LIN {X 0,Y 593.87,Z 557.03,A -85,B 0,C 180,E1 1454.349,E2 1454.349} C_VEL
LIN {X 0,Y 593.894,Z 557.03,A -85,B 0,C 180,E1 1459.392,E2 1459.392} C_VEL
LIN {X 0,Y 593.837,Z 557.03,A -85,B 0,C 180,E1 1464.073,E2 1464.073} C_VEL
LIN {X 0,Y 593.773,Z 557.03,A -85,B 0,C 180,E1 1468.976,E2 1468.976} C_VEL
LIN {X 0,Y 593.884,Z 557.03,A -85,B 0,C 180,E1 1474.113,E2 1474.113} C_VEL
LIN {X 0,Y 593.674,Z 557.03,A -85,B 0,C 180,E1 1480.084,E2 1480.084} C_VEL
LIN {X 0,Y 593.805,Z 557.03,A -85,B 0,C 180,E1 1485.551,E2 1485.551} C_VEL
LIN {X 0,Y 593.737,Z 557.03,A -85,B 0,C 180,E1 1490.393,E2 1490.393} C_VEL
LIN {X 0,Y 593.676,Z 557.03,A -85,B 0,C 180,E1 1495.87,E2 1495.87} C_VEL
LIN {X 0,Y 593.712,Z 557.03,A -85,B 0,C 180,E1 1501.018,E2 1501.018} C_VEL
LIN {X 0,Y 594.01,Z 557.03,A -85,B 0,C 180,E1 1504.046,E2 1504.046} C_VEL
LIN {X 0,Y 596.269,Z 566.972,A -85,B 0,C 180,E1 1504.292,E2 1504.292} C_VEL
LIN {X 0,Y 596.144,Z 608.591,A -85,B 0,C 180,E1 1505.004,E2 1505.004} C_VEL
LIN {X 0,Y 595.921,Z 644.674,A -85,B 0,C 180,E1 1506.196,E2 1506.196} C_VEL
LIN {X 0,Y 595.546,Z 679.968,A -85,B 0,C 180,E1 1507.979,E2 1507.979} C_VEL
LIN {X 0,Y 595.091,Z 712.148,A -85,B 0,C 180,E1 1510.27,E2 1510.27} C_VEL
LIN {X 0,Y 594.695,Z 739.802,A -85,B 0,C 180,E1 1512.909,E2 1512.909} C_VEL
LIN {X 0,Y 594.485,Z 763.471,A -85,B 0,C 180,E1 1515.907,E2 1515.907} C_VEL
LIN {X 0,Y 594.288,Z 782.426,A -85,B 0,C 180,E1 1519.194,E2 1519.194} C_VEL
LIN {X 0,Y 594.237,Z 796.245,A -85,B 0,C 180,E1 1522.681,E2 1522.681} C_VEL
LIN {X 0,Y 594.179,Z 803.544,A -85,B 0,C 180,E1 1525.616,E2 1525.616} C_VEL
LIN {X 0,Y 594.18,Z 807.038,A -85,B 0,C 180,E1 1528.54,E2 1528.54} C_VEL
LIN {X 0,Y 594.291,Z 806.976,A -85,B 0,C 180,E1 1531.46,E2 1531.46} C_VEL
LIN {X 0,Y 594.344,Z 801.858,A -85,B 0,C 180,E1 1535.115,E2 1535.115} C_VEL
LIN {X 0,Y 594.313,Z 790.835,A -85,B 0,C 180,E1 1538.792,E2 1538.792} C_VEL
LIN {X 0,Y 594.4,Z 773.951,A -85,B 0,C 180,E1 1542.317,E2 1542.317} C_VEL
LIN {X 0,Y 594.592,Z 752.418,A -85,B 0,C 180,E1 1545.507,E2 1545.507} C_VEL
LIN {X 0,Y 594.939,Z 725.593,A -85,B 0,C 180,E1 1548.452,E2 1548.452} C_VEL
LIN {X 0,Y 595.327,Z 694.534,A -85,B 0,C 180,E1 1550.979,E2 1550.979} C_VEL
LIN {X 0,Y 595.759,Z 661.466,A -85,B 0,C 180,E1 1552.949,E2 1552.949} C_VEL
LIN {X 0,Y 596.16,Z 625.785,A -85,B 0,C 180,E1 1554.413,E2 1554.413} C_VEL
LIN {X 0,Y 596.353,Z 590.481,A -85,B 0,C 180,E1 1555.284,E2 1555.284} C_VEL
LIN {X 0,Y 595.411,Z 561.137,A -85,B 0,C 180,E1 1555.735,E2 1555.735} C_VEL
LIN {X 0,Y 594.246,Z 557.03,A -85,B 0,C 180,E1 1555.896,E2 1555.896} C_VEL
LIN {X 0,Y 593.862,Z 557.03,A -85,B 0,C 180,E1 1562.725,E2 1562.725} C_VEL
LIN {X 0,Y 593.696,Z 557.03,A -85,B 0,C 180,E1 1567.767,E2 1567.767} C_VEL
LIN {X 0,Y 593.717,Z 557.03,A -85,B 0,C 180,E1 1573.514,E2 1573.514} C_VEL
LIN {X 0,Y 593.8,Z 557.03,A -85,B 0,C 180,E1 1578.48,E2 1578.48} C_VEL
LIN {X 0,Y 593.827,Z 557.03,A -85,B 0,C 180,E1 1584.675,E2 1584.675} C_VEL
LIN {X 0,Y 593.742,Z 557.03,A -85,B 0,C 180,E1 1591.023,E2 1591.023} C_VEL
LIN {X 0,Y 593.928,Z 557.03,A -85,B 0,C 180,E1 1595.931,E2 1595.931} C_VEL
LIN {X 0,Y 594.027,Z 557.03,A -85,B 0,C 180,E1 1600.651,E2 1600.651} C_VEL
LIN {X 0,Y 594.189,Z 557.03,A -85,B 0,C 180,E1 1606.744,E2 1606.744} C_VEL
LIN {X 0,Y 593.995,Z 557.03,A -85,B 0,C 180,E1 1612.679,E2 1612.679} C_VEL
LIN {X 0,Y 593.974,Z 557.03,A -85,B 0,C 180,E1 1617.639,E2 1617.639} C_VEL
LIN {X 0,Y 594.086,Z 557.03,A -85,B 0,C 180,E1 1620.924,E2 1620.924} C_VEL
LIN {X 0,Y 591.572,Z 557.03,A -85,B 0,C 180,E1 1622.168,E2 1622.168} C_VEL
LIN {X 0,Y 586.053,Z 557.03,A -85,B 0,C 180,E1 1624.028,E2 1624.028} C_VEL
LIN {X 0,Y 585.975,Z 557.03,A -85,B 0,C 180,E1 1624.243,E2 1624.243} C_VEL
LIN {X 0,Y 585.921,Z 557.03,A -85,B 0,C 180,E1 1628.919,E2 1628.919} C_VEL
LIN {X 0,Y 585.911,Z 557.03,A -85,B 0,C 180,E1 1633.448,E2 1633.448} C_VEL
LIN {X 0,Y 585.999,Z 557.03,A -85,B 0,C 180,E1 1639.625,E2 1639.625} C_VEL
LIN {X 0,Y 585.974,Z 557.03,A -85,B 0,C 180,E1 1646.054,E2 1646.054} C_VEL
LIN {X 0,Y 585.817,Z 557.03,A -85,B 0,C 180,E1 1651.473,E2 1651.473} C_VEL
LIN {X 0,Y 585.878,Z 557.03,A -85,B 0,C 180,E1 1656.764,E2 1656.764} C_VEL
LIN {X 0,Y 585.916,Z 557.03,A -85,B 0,C 180,E1 1662.207,E2 1662.207} C_VEL
LIN {X 0,Y 585.735,Z 557.03,A -85,B 0,C 180,E1 1667.774,E2 1667.774} C_VEL
LIN {X 0,Y 585.716,Z 557.03,A -85,B 0,C 180,E1 1673.253,E2 1673.253} C_VEL
LIN {X 0,Y 586.076,Z 557.03,A -85,B 0,C 180,E1 1678.48,E2 1678.48} C_VEL
LIN {X 0,Y 586.167,Z 557.03,A -85,B 0,C 180,E1 1679.281,E2 1679.281} C_VEL
LIN {X 0,Y 589.705,Z 569.159,A -85,B 0,C 180,E1 1679.677,E2 1679.677} C_VEL
LIN {X 0,Y 589.901,Z 625.835,A -85,B 0,C 180,E1 1680.633,E2 1680.633} C_VEL
LIN {X 0,Y 589.42,Z 664.732,A -85,B 0,C 180,E1 1681.888,E2 1681.888} C_VEL
LIN {X 0,Y 588.759,Z 703.392,A -85,B 0,C 180,E1 1683.792,E2 1683.792} C_VEL
LIN {X 0,Y 588.073,Z 737.237,A -85,B 0,C 180,E1 1686.086,E2 1686.086} C_VEL
LIN {X 0,Y 587.435,Z 768.24,A -85,B 0,C 180,E1 1688.849,E2 1688.849} C_VEL
LIN {X 0,Y 586.926,Z 795.235,A -85,B 0,C 180,E1 1691.968,E2 1691.968} C_VEL
LIN {X 0,Y 586.625,Z 817.633,A -85,B 0,C 180,E1 1695.35,E2 1695.35} C_VEL
LIN {X 0,Y 586.421,Z 834.783,A -85,B 0,C 180,E1 1698.825,E2 1698.825} C_VEL
LIN {X 0,Y 586.319,Z 847.614,A -85,B 0,C 180,E1 1702.582,E2 1702.582} C_VEL
LIN {X 0,Y 586.252,Z 853.933,A -85,B 0,C 180,E1 1705.557,E2 1705.557} C_VEL
LIN {X 0,Y 586.272,Z 857.083,A -85,B 0,C 180,E1 1708.52,E2 1708.52} C_VEL
LIN {X 0,Y 586.393,Z 857.083,A -85,B 0,C 180,E1 1711.48,E2 1711.48} C_VEL
LIN {X 0,Y 586.488,Z 852.725,A -85,B 0,C 180,E1 1715.184,E2 1715.184} C_VEL
LIN {X 0,Y 586.432,Z 841.96,A -85,B 0,C 180,E1 1719.286,E2 1719.286} C_VEL
LIN {X 0,Y 586.556,Z 826.221,A -85,B 0,C 180,E1 1723.054,E2 1723.054} C_VEL
LIN {X 0,Y 586.778,Z 804.806,A -85,B 0,C 180,E1 1726.703,E2 1726.703} C_VEL
LIN {X 0,Y 587.203,Z 779.518,A -85,B 0,C 180,E1 1729.947,E2 1729.947} C_VEL
LIN {X 0,Y 587.792,Z 749.839,A -85,B 0,C 180,E1 1732.877,E2 1732.877} C_VEL
LIN {X 0,Y 588.471,Z 716.378,A -85,B 0,C 180,E1 1735.404,E2 1735.404} C_VEL
LIN {X 0,Y 589.168,Z 681.902,A -85,B 0,C 180,E1 1737.348,E2 1737.348} C_VEL
LIN {X 0,Y 589.721,Z 644.987,A -85,B 0,C 180,E1 1738.821,E2 1738.821} C_VEL
LIN {X 0,Y 590.083,Z 607.015,A -85,B 0,C 180,E1 1739.755,E2 1739.755} C_VEL
LIN {X 0,Y 589.2,Z 565.193,A -85,B 0,C 180,E1 1740.406,E2 1740.406} C_VEL
LIN {X 0,Y 586.163,Z 557.03,A -85,B 0,C 180,E1 1740.72,E2 1740.72} C_VEL
LIN {X 0,Y 585.92,Z 557.03,A -85,B 0,C 180,E1 1744.646,E2 1744.646} C_VEL
LIN {X 0,Y 585.784,Z 557.03,A -85,B 0,C 180,E1 1750.253,E2 1750.253} C_VEL
LIN {X 0,Y 585.931,Z 557.03,A -85,B 0,C 180,E1 1756.346,E2 1756.346} C_VEL
LIN {X 0,Y 585.851,Z 557.03,A -85,B 0,C 180,E1 1761.669,E2 1761.669} C_VEL
LIN {X 0,Y 585.745,Z 557.03,A -85,B 0,C 180,E1 1767.127,E2 1767.127} C_VEL
LIN {X 0,Y 585.781,Z 557.03,A -85,B 0,C 180,E1 1772.276,E2 1772.276} C_VEL
LIN {X 0,Y 585.838,Z 557.03,A -85,B 0,C 180,E1 1777.192,E2 1777.192} C_VEL
LIN {X 0,Y 586.065,Z 557.03,A -85,B 0,C 180,E1 1781.941,E2 1781.941} C_VEL
LIN {X 0,Y 585.802,Z 557.03,A -85,B 0,C 180,E1 1788.068,E2 1788.068} C_VEL
LIN {X 0,Y 586.302,Z 557.03,A -85,B 0,C 180,E1 1794.071,E2 1794.071} C_VEL
LIN {X 0,Y 586.079,Z 557.03,A -85,B 0,C 180,E1 1800,E2 1800} C_VEL
LIN {X 0,Y 586.146,Z 557.03,A -85,B 0,C 180,E1 1804.444,E2 1804.444} C_VEL
LIN {X 0,Y 586.134,Z 557.03,A -85,B 0,C 180,E1 1808.915,E2 1808.915} C_VEL
LIN {X 0,Y 586.16,Z 557.03,A -85,B 0,C 180,E1 1813.441,E2 1813.441} C_VEL
LIN {X 0,Y 586.114,Z 557.03,A -85,B 0,C 180,E1 1818.057,E2 1818.057} C_VEL
LIN {X 0,Y 586.018,Z 557.03,A -85,B 0,C 180,E1 1822.8,E2 1822.8} C_VEL
LIN {X 0,Y 585.848,Z 557.03,A -85,B 0,C 180,E1 1828.515,E2 1828.515} C_VEL
LIN {X 0,Y 585.87,Z 557.03,A -85,B 0,C 180,E1 1834.645,E2 1834.645} C_VEL
LIN {X 0,Y 585.78,Z 557.03,A -85,B 0,C 180,E1 1840.25,E2 1840.25} C_VEL
LIN {X 0,Y 585.931,Z 557.03,A -85,B 0,C 180,E1 1846.341,E2 1846.341} C_VEL
LIN {X 0,Y 585.838,Z 557.03,A -85,B 0,C 180,E1 1851.665,E2 1851.665} C_VEL
LIN {X 0,Y 585.75,Z 557.03,A -85,B 0,C 180,E1 1857.125,E2 1857.125} C_VEL
LIN {X 0,Y 585.761,Z 557.03,A -85,B 0,C 180,E1 1862.273,E2 1862.273} C_VEL
LIN {X 0,Y 586.006,Z 557.03,A -85,B 0,C 180,E1 1863.668,E2 1863.668} C_VEL
LIN {X 0,Y 589.166,Z 566.473,A -85,B 0,C 180,E1 1863.953,E2 1863.953} C_VEL
LIN {X 0,Y 588.944,Z 609.999,A -85,B 0,C 180,E1 1864.714,E2 1864.714} C_VEL
LIN {X 0,Y 588.628,Z 645.318,A -85,B 0,C 180,E1 1865.91,E2 1865.91} C_VEL
LIN {X 0,Y 588.083,Z 681.056,A -85,B 0,C 180,E1 1867.754,E2 1867.754} C_VEL
LIN {X 0,Y 587.533,Z 712.143,A -85,B 0,C 180,E1 1870.006,E2 1870.006} C_VEL
LIN {X 0,Y 586.988,Z 740.443,A -85,B 0,C 180,E1 1872.749,E2 1872.749} C_VEL
LIN {X 0,Y 586.655,Z 764.995,A -85,B 0,C 180,E1 1875.953,E2 1875.953} C_VEL
LIN {X 0,Y 586.432,Z 783.104,A -85,B 0,C 180,E1 1879.194,E2 1879.194} C_VEL
LIN {X 0,Y 586.347,Z 796.243,A -85,B 0,C 180,E1 1882.582,E2 1882.582} C_VEL
LIN {X 0,Y 586.284,Z 803.542,A -85,B 0,C 180,E1 1885.556,E2 1885.556} C_VEL
LIN {X 0,Y 586.287,Z 807.038,A -85,B 0,C 180,E1 1888.52,E2 1888.52} C_VEL
LIN {X 0,Y 586.387,Z 806.977,A -85,B 0,C 180,E1 1891.479,E2 1891.479} C_VEL
LIN {X 0,Y 586.451,Z 801.86,A -85,B 0,C 180,E1 1895.184,E2 1895.184} C_VEL
LIN {X 0,Y 586.417,Z 790.837,A -85,B 0,C 180,E1 1898.911,E2 1898.911} C_VEL
LIN {X 0,Y 586.555,Z 775.044,A -85,B 0,C 180,E1 1902.295,E2 1902.295} C_VEL
LIN {X 0,Y 586.815,Z 753.892,A -85,B 0,C 180,E1 1905.526,E2 1905.526} C_VEL
LIN {X 0,Y 587.241,Z 728.56,A -85,B 0,C 180,E1 1908.411,E2 1908.411} C_VEL
LIN {X 0,Y 587.784,Z 697.258,A -85,B 0,C 180,E1 1911.066,E2 1911.066} C_VEL
LIN {X 0,Y 588.325,Z 664.502,A -85,B 0,C 180,E1 1913.095,E2 1913.095} C_VEL
LIN {X 0,Y 588.832,Z 630.553,A -85,B 0,C 180,E1 1914.568,E2 1914.568} C_VEL
LIN {X 0,Y 589.213,Z 592.616,A -85,B 0,C 180,E1 1915.576,E2 1915.576} C_VEL
LIN {X 0,Y 588.439,Z 563.817,A -85,B 0,C 180,E1 1916.027,E2 1916.027} C_VEL
LIN {X 0,Y 586.319,Z 557.03,A -85,B 0,C 180,E1 1916.265,E2 1916.265} C_VEL
LIN {X 0,Y 585.961,Z 557.03,A -85,B 0,C 180,E1 1922.861,E2 1922.861} C_VEL
LIN {X 0,Y 585.789,Z 557.03,A -85,B 0,C 180,E1 1929.165,E2 1929.165} C_VEL
LIN {X 0,Y 585.863,Z 557.03,A -85,B 0,C 180,E1 1934.247,E2 1934.247} C_VEL
LIN {X 0,Y 585.851,Z 557.03,A -85,B 0,C 180,E1 1939.756,E2 1939.756} C_VEL
LIN {X 0,Y 585.812,Z 557.03,A -85,B 0,C 180,E1 1945.351,E2 1945.351} C_VEL
LIN {X 0,Y 585.868,Z 557.03,A -85,B 0,C 180,E1 1950.595,E2 1950.595} C_VEL
LIN {X 0,Y 585.999,Z 557.03,A -85,B 0,C 180,E1 1955.584,E2 1955.584} C_VEL
LIN {X 0,Y 586.117,Z 557.03,A -85,B 0,C 180,E1 1960.38,E2 1960.38} C_VEL
LIN {X 0,Y 586.263,Z 557.03,A -85,B 0,C 180,E1 1966.561,E2 1966.561} C_VEL
LIN {X 0,Y 586.091,Z 557.03,A -85,B 0,C 180,E1 1972.579,E2 1972.579} C_VEL
LIN {X 0,Y 586.226,Z 557.03,A -85,B 0,C 180,E1 1977.04,E2 1977.04} C_VEL
LIN {X 0,Y 586.312,Z 557.03,A -85,B 0,C 180,E1 1981.48,E2 1981.48} C_VEL
LIN {X 0,Y 585.975,Z 557.03,A -85,B 0,C 180,E1 1984.243,E2 1984.243} C_VEL
LIN {X 0,Y 583.549,Z 557.03,A -85,B 0,C 180,E1 1985.506,E2 1985.506} C_VEL
LIN {X 0,Y 578.046,Z 557.03,A -85,B 0,C 180,E1 1987.615,E2 1987.615} C_VEL
LIN {X 0,Y 578.057,Z 557.03,A -85,B 0,C 180,E1 1992.095,E2 1992.095} C_VEL
LIN {X 0,Y 577.989,Z 557.03,A -85,B 0,C 180,E1 1996.746,E2 1996.746} C_VEL
LIN {X 0,Y 578.036,Z 557.03,A -85,B 0,C 180,E1 2001.511,E2 2001.511} C_VEL
LIN {X 0,Y 577.918,Z 557.03,A -85,B 0,C 180,E1 2007.034,E2 2007.034} C_VEL
LIN {X 0,Y 577.909,Z 557.03,A -85,B 0,C 180,E1 2011.597,E2 2011.597} C_VEL
LIN {X 0,Y 577.961,Z 557.03,A -85,B 0,C 180,E1 2017.048,E2 2017.048} C_VEL
LIN {X 0,Y 577.992,Z 557.03,A -85,B 0,C 180,E1 2022.924,E2 2022.924} C_VEL
LIN {X 0,Y 577.831,Z 557.03,A -85,B 0,C 180,E1 2029.076,E2 2029.076} C_VEL
LIN {X 0,Y 577.894,Z 557.03,A -85,B 0,C 180,E1 2034.803,E2 2034.803} C_VEL
LIN {X 0,Y 578.209,Z 557.03,A -85,B 0,C 180,E1 2038.834,E2 2038.834} C_VEL
LIN {X 0,Y 582.926,Z 570.487,A -85,B 0,C 180,E1 2039.305,E2 2039.305} C_VEL
LIN {X 0,Y 582.993,Z 625.619,A -85,B 0,C 180,E1 2040.244,E2 2040.244} C_VEL
LIN {X 0,Y 582.368,Z 664.477,A -85,B 0,C 180,E1 2041.506,E2 2041.506} C_VEL
LIN {X 0,Y 581.597,Z 701.682,A -85,B 0,C 180,E1 2043.339,E2 2043.339} C_VEL
LIN {X 0,Y 580.656,Z 737.538,A -85,B 0,C 180,E1 2045.786,E2 2045.786} C_VEL
LIN {X 0,Y 579.842,Z 768.239,A -85,B 0,C 180,E1 2048.558,E2 2048.558} C_VEL
LIN {X 0,Y 579.211,Z 795.236,A -85,B 0,C 180,E1 2051.719,E2 2051.719} C_VEL
LIN {X 0,Y 578.817,Z 817.891,A -85,B 0,C 180,E1 2055.193,E2 2055.193} C_VEL
LIN {X 0,Y 578.527,Z 834.783,A -85,B 0,C 180,E1 2058.67,E2 2058.67} C_VEL
LIN {X 0,Y 578.432,Z 847.614,A -85,B 0,C 180,E1 2062.48,E2 2062.48} C_VEL
LIN {X 0,Y 578.352,Z 853.933,A -85,B 0,C 180,E1 2065.496,E2 2065.496} C_VEL
LIN {X 0,Y 578.372,Z 857.083,A -85,B 0,C 180,E1 2068.5,E2 2068.5} C_VEL
LIN {X 0,Y 578.487,Z 857.083,A -85,B 0,C 180,E1 2071.5,E2 2071.5} C_VEL
LIN {X 0,Y 578.588,Z 852.751,A -85,B 0,C 180,E1 2075.24,E2 2075.24} C_VEL
LIN {X 0,Y 578.536,Z 843.209,A -85,B 0,C 180,E1 2079.034,E2 2079.034} C_VEL
LIN {X 0,Y 578.709,Z 828.079,A -85,B 0,C 180,E1 2082.849,E2 2082.849} C_VEL
LIN {X 0,Y 578.986,Z 806.282,A -85,B 0,C 180,E1 2086.718,E2 2086.718} C_VEL
LIN {X 0,Y 579.54,Z 779.914,A -85,B 0,C 180,E1 2090.177,E2 2090.177} C_VEL
LIN {X 0,Y 580.333,Z 750.003,A -85,B 0,C 180,E1 2093.174,E2 2093.174} C_VEL
LIN {X 0,Y 581.147,Z 716.949,A -85,B 0,C 180,E1 2095.709,E2 2095.709} C_VEL
LIN {X 0,Y 582.032,Z 682.321,A -85,B 0,C 180,E1 2097.691,E2 2097.691} C_VEL
LIN {X 0,Y 582.745,Z 645.845,A -85,B 0,C 180,E1 2099.171,E2 2099.171} C_VEL
LIN {X 0,Y 583.207,Z 608.121,A -85,B 0,C 180,E1 2100.124,E2 2100.124} C_VEL
LIN {X 0,Y 582.48,Z 567.885,A -85,B 0,C 180,E1 2100.757,E2 2100.757} C_VEL
LIN {X 0,Y 578.206,Z 557.03,A -85,B 0,C 180,E1 2101.237,E2 2101.237} C_VEL
LIN {X 0,Y 577.815,Z 557.03,A -85,B 0,C 180,E1 2107.062,E2 2107.062} C_VEL
LIN {X 0,Y 577.865,Z 557.03,A -85,B 0,C 180,E1 2112.939,E2 2112.939} C_VEL
LIN {X 0,Y 577.973,Z 557.03,A -85,B 0,C 180,E1 2119.091,E2 2119.091} C_VEL
LIN {X 0,Y 577.863,Z 557.03,A -85,B 0,C 180,E1 2124.804,E2 2124.804} C_VEL
LIN {X 0,Y 577.92,Z 557.03,A -85,B 0,C 180,E1 2130.15,E2 2130.15} C_VEL
LIN {X 0,Y 578.072,Z 557.03,A -85,B 0,C 180,E1 2135.226,E2 2135.226} C_VEL
LIN {X 0,Y 578.16,Z 557.03,A -85,B 0,C 180,E1 2140.519,E2 2140.519} C_VEL
LIN {X 0,Y 577.915,Z 557.03,A -85,B 0,C 180,E1 2144.813,E2 2144.813} C_VEL
LIN {X 0,Y 578.044,Z 557.03,A -85,B 0,C 180,E1 2150.959,E2 2150.959} C_VEL
LIN {X 0,Y 578.108,Z 557.03,A -85,B 0,C 180,E1 2155.494,E2 2155.494} C_VEL
LIN {X 0,Y 578.179,Z 557.03,A -85,B 0,C 180,E1 2160,E2 2160} C_VEL
LIN {X 0,Y 578.231,Z 557.03,A -85,B 0,C 180,E1 2164.505,E2 2164.505} C_VEL
LIN {X 0,Y 578.2,Z 557.03,A -85,B 0,C 180,E1 2169.038,E2 2169.038} C_VEL
LIN {X 0,Y 578.061,Z 557.03,A -85,B 0,C 180,E1 2174.28,E2 2174.28} C_VEL
LIN {X 0,Y 578.057,Z 557.03,A -85,B 0,C 180,E1 2179.905,E2 2179.905} C_VEL
LIN {X 0,Y 577.963,Z 557.03,A -85,B 0,C 180,E1 2184.778,E2 2184.778} C_VEL
LIN {X 0,Y 577.835,Z 557.03,A -85,B 0,C 180,E1 2190.154,E2 2190.154} C_VEL
LIN {X 0,Y 577.852,Z 557.03,A -85,B 0,C 180,E1 2195.197,E2 2195.197} C_VEL
LIN {X 0,Y 577.823,Z 557.03,A -85,B 0,C 180,E1 2200.921,E2 2200.921} C_VEL
LIN {X 0,Y 577.979,Z 557.03,A -85,B 0,C 180,E1 2207.174,E2 2207.174} C_VEL
LIN {X 0,Y 577.949,Z 557.03,A -85,B 0,C 180,E1 2212.948,E2 2212.948} C_VEL
LIN {X 0,Y 577.912,Z 557.03,A -85,B 0,C 180,E1 2218.401,E2 2218.401} C_VEL
LIN {X 0,Y 578.048,Z 557.03,A -85,B 0,C 180,E1 2223.282,E2 2223.282} C_VEL
LIN {X 0,Y 582.088,Z 569.469,A -85,B 0,C 180,E1 2223.653,E2 2223.653} C_VEL
LIN {X 0,Y 581.766,Z 611.358,A -85,B 0,C 180,E1 2224.416,E2 2224.416} C_VEL
LIN {X 0,Y 581.322,Z 648.273,A -85,B 0,C 180,E1 2225.714,E2 2225.714} C_VEL
LIN {X 0,Y 580.636,Z 682.224,A -85,B 0,C 180,E1 2227.531,E2 2227.531} C_VEL
LIN {X 0,Y 579.89,Z 714.525,A -85,B 0,C 180,E1 2229.939,E2 2229.939} C_VEL
LIN {X 0,Y 579.241,Z 742.179,A -85,B 0,C 180,E1 2232.706,E2 2232.706} C_VEL
LIN {X 0,Y 578.832,Z 765.779,A -85,B 0,C 180,E1 2235.885,E2 2235.885} C_VEL
LIN {X 0,Y 578.591,Z 783.102,A -85,B 0,C 180,E1 2239.046,E2 2239.046} C_VEL
LIN {X 0,Y 578.46,Z 796.241,A -85,B 0,C 180,E1 2242.48,E2 2242.48} C_VEL
LIN {X 0,Y 578.391,Z 803.541,A -85,B 0,C 180,E1 2245.496,E2 2245.496} C_VEL
LIN {X 0,Y 578.386,Z 807.038,A -85,B 0,C 180,E1 2248.5,E2 2248.5} C_VEL
LIN {X 0,Y 578.482,Z 806.977,A -85,B 0,C 180,E1 2251.499,E2 2251.499} C_VEL
LIN {X 0,Y 578.557,Z 801.862,A -85,B 0,C 180,E1 2255.255,E2 2255.255} C_VEL
LIN {X 0,Y 578.532,Z 790.839,A -85,B 0,C 180,E1 2259.034,E2 2259.034} C_VEL
LIN {X 0,Y 578.706,Z 775.047,A -85,B 0,C 180,E1 2262.465,E2 2262.465} C_VEL
LIN {X 0,Y 579.054,Z 753.898,A -85,B 0,C 180,E1 2265.74,E2 2265.74} C_VEL
LIN {X 0,Y 579.571,Z 728.565,A -85,B 0,C 180,E1 2268.664,E2 2268.664} C_VEL
LIN {X 0,Y 580.256,Z 697.646,A -85,B 0,C 180,E1 2271.325,E2 2271.325} C_VEL
LIN {X 0,Y 580.981,Z 664.452,A -85,B 0,C 180,E1 2273.408,E2 2273.408} C_VEL
LIN {X 0,Y 581.62,Z 630.57,A -85,B 0,C 180,E1 2274.894,E2 2274.894} C_VEL
LIN {X 0,Y 582.084,Z 593.433,A -85,B 0,C 180,E1 2275.896,E2 2275.896} C_VEL
LIN {X 0,Y 581.173,Z 565.297,A -85,B 0,C 180,E1 2276.358,E2 2276.358} C_VEL
LIN {X 0,Y 578.366,Z 557.03,A -85,B 0,C 180,E1 2276.682,E2 2276.682} C_VEL
LIN {X 0,Y 578.03,Z 557.03,A -85,B 0,C 180,E1 2283.371,E2 2283.371} C_VEL
LIN {X 0,Y 577.872,Z 557.03,A -85,B 0,C 180,E1 2288.962,E2 2288.962} C_VEL
LIN {X 0,Y 577.938,Z 557.03,A -85,B 0,C 180,E1 2295.018,E2 2295.018} C_VEL
LIN {X 0,Y 577.903,Z 557.03,A -85,B 0,C 180,E1 2301.044,E2 2301.044} C_VEL
LIN {X 0,Y 577.826,Z 557.03,A -85,B 0,C 180,E1 2306.98,E2 2306.98} C_VEL
LIN {X 0,Y 577.899,Z 557.03,A -85,B 0,C 180,E1 2311.865,E2 2311.865} C_VEL
LIN {X 0,Y 577.97,Z 557.03,A -85,B 0,C 180,E1 2316.864,E2 2316.864} C_VEL
LIN {X 0,Y 578.127,Z 557.03,A -85,B 0,C 180,E1 2321.685,E2 2321.685} C_VEL
LIN {X 0,Y 578.319,Z 557.03,A -85,B 0,C 180,E1 2326.373,E2 2326.373} C_VEL
LIN {X 0,Y 578.191,Z 557.03,A -85,B 0,C 180,E1 2332.477,E2 2332.477} C_VEL
LIN {X 0,Y 578.319,Z 557.03,A -85,B 0,C 180,E1 2336.999,E2 2336.999} C_VEL
LIN {X 0,Y 578.402,Z 557.03,A -85,B 0,C 180,E1 2341.5,E2 2341.5} C_VEL
LIN {X 0,Y 578.359,Z 557.03,A -85,B 0,C 180,E1 2346.011,E2 2346.011} C_VEL
LIN {X 0,Y 578.046,Z 557.03,A -85,B 0,C 180,E1 2347.615,E2 2347.615} C_VEL
LIN {X 0,Y 574.164,Z 557.03,A -85,B 0,C 180,E1 2349.307,E2 2349.307} C_VEL
LIN {X 0,Y 570.229,Z 557.03,A -85,B 0,C 180,E1 2351.022,E2 2351.022} C_VEL
LIN {X 0,Y 570.045,Z 557.03,A -85,B 0,C 180,E1 2357.028,E2 2357.028} C_VEL
LIN {X 0,Y 570.104,Z 557.03,A -85,B 0,C 180,E1 2361.826,E2 2361.826} C_VEL
LIN {X 0,Y 570.047,Z 557.03,A -85,B 0,C 180,E1 2366.84,E2 2366.84} C_VEL
LIN {X 0,Y 569.964,Z 557.03,A -85,B 0,C 180,E1 2372.09,E2 2372.09} C_VEL
LIN {X 0,Y 570.047,Z 557.03,A -85,B 0,C 180,E1 2377.651,E2 2377.651} C_VEL
LIN {X 0,Y 569.989,Z 557.03,A -85,B 0,C 180,E1 2383.677,E2 2383.677} C_VEL
LIN {X 0,Y 569.869,Z 557.03,A -85,B 0,C 180,E1 2388.379,E2 2388.379} C_VEL
LIN {X 0,Y 569.94,Z 557.03,A -85,B 0,C 180,E1 2394.237,E2 2394.237} C_VEL
LIN {X 0,Y 570.269,Z 557.119,A -85,B 0,C 180,E1 2398.354,E2 2398.354} C_VEL
LIN {X 0,Y 576.24,Z 572.825,A -85,B 0,C 180,E1 2398.943,E2 2398.943} C_VEL
LIN {X 0,Y 576.089,Z 626.469,A -85,B 0,C 180,E1 2399.874,E2 2399.874} C_VEL
LIN {X 0,Y 575.334,Z 664.66,A -85,B 0,C 180,E1 2401.133,E2 2401.133} C_VEL
LIN {X 0,Y 574.371,Z 702.616,A -85,B 0,C 180,E1 2403.035,E2 2403.035} C_VEL
LIN {X 0,Y 573.29,Z 737.534,A -85,B 0,C 180,E1 2405.454,E2 2405.454} C_VEL
LIN {X 0,Y 572.246,Z 768.239,A -85,B 0,C 180,E1 2408.259,E2 2408.259} C_VEL
LIN {X 0,Y 571.507,Z 795.238,A -85,B 0,C 180,E1 2411.464,E2 2411.464} C_VEL
LIN {X 0,Y 571.005,Z 817.891,A -85,B 0,C 180,E1 2414.986,E2 2414.986} C_VEL
LIN {X 0,Y 570.684,Z 835.84,A -85,B 0,C 180,E1 2418.777,E2 2418.777} C_VEL
LIN {X 0,Y 570.544,Z 847.614,A -85,B 0,C 180,E1 2422.376,E2 2422.376} C_VEL
LIN {X 0,Y 570.481,Z 853.933,A -85,B 0,C 180,E1 2425.434,E2 2425.434} C_VEL
LIN {X 0,Y 570.483,Z 857.083,A -85,B 0,C 180,E1 2428.479,E2 2428.479} C_VEL
LIN {X 0,Y 570.587,Z 857.083,A -85,B 0,C 180,E1 2431.521,E2 2431.521} C_VEL
LIN {X 0,Y 570.697,Z 852.942,A -85,B 0,C 180,E1 2435.194,E2 2435.194} C_VEL
LIN {X 0,Y 570.649,Z 843.209,A -85,B 0,C 180,E1 2439.16,E2 2439.16} C_VEL
LIN {X 0,Y 570.872,Z 828.08,A -85,B 0,C 180,E1 2443.029,E2 2443.029} C_VEL
LIN {X 0,Y 571.234,Z 806.281,A -85,B 0,C 180,E1 2446.951,E2 2446.951} C_VEL
LIN {X 0,Y 571.882,Z 781,A -85,B 0,C 180,E1 2450.334,E2 2450.334} C_VEL
LIN {X 0,Y 572.811,Z 751.529,A -85,B 0,C 180,E1 2453.359,E2 2453.359} C_VEL
LIN {X 0,Y 573.817,Z 718.542,A -85,B 0,C 180,E1 2455.952,E2 2455.952} C_VEL
LIN {X 0,Y 574.934,Z 682.748,A -85,B 0,C 180,E1 2458.042,E2 2458.042} C_VEL
LIN {X 0,Y 575.793,Z 646.2,A -85,B 0,C 180,E1 2459.546,E2 2459.546} C_VEL
LIN {X 0,Y 576.376,Z 607.896,A -85,B 0,C 180,E1 2460.522,E2 2460.522} C_VEL
LIN {X 0,Y 575.816,Z 570.4,A -85,B 0,C 180,E1 2461.117,E2 2461.117} C_VEL
LIN {X 0,Y 570.272,Z 557.03,A -85,B 0,C 180,E1 2461.709,E2 2461.709} C_VEL
LIN {X 0,Y 569.911,Z 557.03,A -85,B 0,C 180,E1 2467.664,E2 2467.664} C_VEL
LIN {X 0,Y 569.909,Z 557.03,A -85,B 0,C 180,E1 2473.688,E2 2473.688} C_VEL
LIN {X 0,Y 570.008,Z 557.03,A -85,B 0,C 180,E1 2478.394,E2 2478.394} C_VEL
LIN {X 0,Y 569.984,Z 557.03,A -85,B 0,C 180,E1 2484.243,E2 2484.243} C_VEL
LIN {X 0,Y 570.024,Z 557.03,A -85,B 0,C 180,E1 2489.693,E2 2489.693} C_VEL
LIN {X 0,Y 570.11,Z 557.03,A -85,B 0,C 180,E1 2494.856,E2 2494.856} C_VEL
LIN {X 0,Y 570.188,Z 557.03,A -85,B 0,C 180,E1 2499.807,E2 2499.807} C_VEL
LIN {X 0,Y 570.027,Z 557.03,A -85,B 0,C 180,E1 2504.598,E2 2504.598} C_VEL
LIN {X 0,Y 570.14,Z 557.03,A -85,B 0,C 180,E1 2510.832,E2 2510.832} C_VEL
LIN {X 0,Y 570.23,Z 557.03,A -85,B 0,C 180,E1 2515.431,E2 2515.431} C_VEL
LIN {X 0,Y 570.292,Z 557.03,A -85,B 0,C 180,E1 2520,E2 2520} C_VEL
LIN {X 0,Y 570.329,Z 557.03,A -85,B 0,C 180,E1 2524.567,E2 2524.567} C_VEL
LIN {X 0,Y 570.27,Z 557.03,A -85,B 0,C 180,E1 2529.165,E2 2529.165} C_VEL
LIN {X 0,Y 570.265,Z 557.03,A -85,B 0,C 180,E1 2533.823,E2 2533.823} C_VEL
LIN {X 0,Y 570.232,Z 557.03,A -85,B 0,C 180,E1 2538.578,E2 2538.578} C_VEL
LIN {X 0,Y 570.142,Z 557.03,A -85,B 0,C 180,E1 2543.472,E2 2543.472} C_VEL
LIN {X 0,Y 569.989,Z 557.03,A -85,B 0,C 180,E1 2548.768,E2 2548.768} C_VEL
LIN {X 0,Y 569.949,Z 557.03,A -85,B 0,C 180,E1 2554.562,E2 2554.562} C_VEL
LIN {X 0,Y 569.919,Z 557.03,A -85,B 0,C 180,E1 2559.608,E2 2559.608} C_VEL
LIN {X 0,Y 569.973,Z 557.03,A -85,B 0,C 180,E1 2565.821,E2 2565.821} C_VEL
LIN {X 0,Y 570.011,Z 557.03,A -85,B 0,C 180,E1 2570.395,E2 2570.395} C_VEL
LIN {X 0,Y 569.891,Z 557.03,A -85,B 0,C 180,E1 2576.088,E2 2576.088} C_VEL
LIN {X 0,Y 569.928,Z 557.03,A -85,B 0,C 180,E1 2581.433,E2 2581.433} C_VEL
LIN {X 0,Y 570.127,Z 557.856,A -85,B 0,C 180,E1 2582.896,E2 2582.896} C_VEL
LIN {X 0,Y 575.03,Z 572.151,A -85,B 0,C 180,E1 2583.341,E2 2583.341} C_VEL
LIN {X 0,Y 574.613,Z 612.99,A -85,B 0,C 180,E1 2584.118,E2 2584.118} C_VEL
LIN {X 0,Y 574.004,Z 650.621,A -85,B 0,C 180,E1 2585.497,E2 2585.497} C_VEL
LIN {X 0,Y 573.175,Z 683.835,A -85,B 0,C 180,E1 2587.33,E2 2587.33} C_VEL
LIN {X 0,Y 572.306,Z 715.702,A -85,B 0,C 180,E1 2589.766,E2 2589.766} C_VEL
LIN {X 0,Y 571.501,Z 743.468,A -85,B 0,C 180,E1 2592.622,E2 2592.622} C_VEL
LIN {X 0,Y 571.032,Z 766.203,A -85,B 0,C 180,E1 2595.757,E2 2595.757} C_VEL
LIN {X 0,Y 570.747,Z 783.333,A -85,B 0,C 180,E1 2598.945,E2 2598.945} C_VEL
LIN {X 0,Y 570.58,Z 796.24,A -85,B 0,C 180,E1 2602.375,E2 2602.375} C_VEL
LIN {X 0,Y 570.526,Z 803.539,A -85,B 0,C 180,E1 2605.433,E2 2605.433} C_VEL
LIN {X 0,Y 570.495,Z 807.038,A -85,B 0,C 180,E1 2608.479,E2 2608.479} C_VEL
LIN {X 0,Y 570.583,Z 806.978,A -85,B 0,C 180,E1 2611.52,E2 2611.52} C_VEL
LIN {X 0,Y 570.669,Z 802.109,A -85,B 0,C 180,E1 2615.207,E2 2615.207} C_VEL
LIN {X 0,Y 570.678,Z 792.181,A -85,B 0,C 180,E1 2618.775,E2 2618.775} C_VEL
LIN {X 0,Y 570.859,Z 776.108,A -85,B 0,C 180,E1 2622.444,E2 2622.444} C_VEL
LIN {X 0,Y 571.255,Z 755.365,A -85,B 0,C 180,E1 2625.763,E2 2625.763} C_VEL
LIN {X 0,Y 571.89,Z 730.536,A -85,B 0,C 180,E1 2628.718,E2 2628.718} C_VEL
LIN {X 0,Y 572.705,Z 700.358,A -85,B 0,C 180,E1 2631.417,E2 2631.417} C_VEL
LIN {X 0,Y 573.584,Z 666.946,A -85,B 0,C 180,E1 2633.592,E2 2633.592} C_VEL
LIN {X 0,Y 574.324,Z 633.261,A -85,B 0,C 180,E1 2635.132,E2 2635.132} C_VEL
LIN {X 0,Y 574.877,Z 597.222,A -85,B 0,C 180,E1 2636.165,E2 2636.165} C_VEL
LIN {X 0,Y 574.433,Z 568.205,A -85,B 0,C 180,E1 2636.653,E2 2636.653} C_VEL
LIN {X 0,Y 570.381,Z 557.03,A -85,B 0,C 180,E1 2637.082,E2 2637.082} C_VEL
LIN {X 0,Y 570.017,Z 557.03,A -85,B 0,C 180,E1 2643.903,E2 2643.903} C_VEL
LIN {X 0,Y 569.929,Z 557.03,A -85,B 0,C 180,E1 2649.615,E2 2649.615} C_VEL
LIN {X 0,Y 569.971,Z 557.03,A -85,B 0,C 180,E1 2655.825,E2 2655.825} C_VEL
LIN {X 0,Y 569.987,Z 557.03,A -85,B 0,C 180,E1 2660.397,E2 2660.397} C_VEL
LIN {X 0,Y 569.883,Z 557.03,A -85,B 0,C 180,E1 2665.446,E2 2665.446} C_VEL
LIN {X 0,Y 569.967,Z 557.03,A -85,B 0,C 180,E1 2671.235,E2 2671.235} C_VEL
LIN {X 0,Y 570.112,Z 557.03,A -85,B 0,C 180,E1 2676.527,E2 2676.527} C_VEL
LIN {X 0,Y 570.227,Z 557.03,A -85,B 0,C 180,E1 2681.422,E2 2681.422} C_VEL
LIN {X 0,Y 570.394,Z 557.03,A -85,B 0,C 180,E1 2686.18,E2 2686.18} C_VEL
LIN {X 0,Y 570.282,Z 557.03,A -85,B 0,C 180,E1 2692.373,E2 2692.373} C_VEL
LIN {X 0,Y 570.411,Z 557.03,A -85,B 0,C 180,E1 2696.957,E2 2696.957} C_VEL
LIN {X 0,Y 570.503,Z 557.03,A -85,B 0,C 180,E1 2701.521,E2 2701.521} C_VEL
LIN {X 0,Y 570.145,Z 557.03,A -85,B 0,C 180,E1 2707.611,E2 2707.611} C_VEL
LIN {X 0,Y 570.229,Z 557.03,A -85,B 0,C 180,E1 2711.022,E2 2711.022} C_VEL
LIN {X 0,Y 566.159,Z 557.03,A -85,B 0,C 180,E1 2712.733,E2 2712.733} C_VEL
LIN {X 0,Y 562.174,Z 557.03,A -85,B 0,C 180,E1 2714.469,E2 2714.469} C_VEL
LIN {X 0,Y 562.22,Z 557.03,A -85,B 0,C 180,E1 2720.492,E2 2720.492} C_VEL
LIN {X 0,Y 562.214,Z 557.03,A -85,B 0,C 180,E1 2725.522,E2 2725.522} C_VEL
LIN {X 0,Y 562.091,Z 557.03,A -85,B 0,C 180,E1 2730.781,E2 2730.781} C_VEL
LIN {X 0,Y 562.098,Z 557.03,A -85,B 0,C 180,E1 2736.338,E2 2736.338} C_VEL
LIN {X 0,Y 562.067,Z 557.03,A -85,B 0,C 180,E1 2742.329,E2 2742.329} C_VEL
LIN {X 0,Y 561.948,Z 557.03,A -85,B 0,C 180,E1 2747.657,E2 2747.657} C_VEL
LIN {X 0,Y 562.024,Z 557.03,A -85,B 0,C 180,E1 2753.913,E2 2753.913} C_VEL
LIN {X 0,Y 562.347,Z 557.399,A -85,B 0,C 180,E1 2757.859,E2 2757.859} C_VEL
LIN {X 0,Y 569.51,Z 574.363,A -85,B 0,C 180,E1 2758.557,E2 2758.557} C_VEL
LIN {X 0,Y 569.283,Z 625.797,A -85,B 0,C 180,E1 2759.457,E2 2759.457} C_VEL
LIN {X 0,Y 568.395,Z 663.192,A -85,B 0,C 180,E1 2760.681,E2 2760.681} C_VEL
LIN {X 0,Y 567.268,Z 701.202,A -85,B 0,C 180,E1 2762.58,E2 2762.58} C_VEL
LIN {X 0,Y 565.926,Z 736.722,A -85,B 0,C 180,E1 2765.045,E2 2765.045} C_VEL
LIN {X 0,Y 564.69,Z 768.239,A -85,B 0,C 180,E1 2767.953,E2 2767.953} C_VEL
LIN {X 0,Y 563.796,Z 795.239,A -85,B 0,C 180,E1 2771.201,E2 2771.201} C_VEL
LIN {X 0,Y 563.194,Z 817.463,A -85,B 0,C 180,E1 2774.694,E2 2774.694} C_VEL
LIN {X 0,Y 562.774,Z 834.827,A -85,B 0,C 180,E1 2778.36,E2 2778.36} C_VEL
LIN {X 0,Y 562.675,Z 847.614,A -85,B 0,C 180,E1 2782.268,E2 2782.268} C_VEL
LIN {X 0,Y 562.579,Z 853.933,A -85,B 0,C 180,E1 2785.369,E2 2785.369} C_VEL
LIN {X 0,Y 562.582,Z 857.083,A -85,B 0,C 180,E1 2788.458,E2 2788.458} C_VEL
LIN {X 0,Y 562.681,Z 857.083,A -85,B 0,C 180,E1 2791.542,E2 2791.542} C_VEL
LIN {X 0,Y 562.757,Z 852.534,A -85,B 0,C 180,E1 2795.505,E2 2795.505} C_VEL
LIN {X 0,Y 562.743,Z 841.959,A -85,B 0,C 180,E1 2799.681,E2 2799.681} C_VEL
LIN {X 0,Y 563.011,Z 826.217,A -85,B 0,C 180,E1 2803.61,E2 2803.61} C_VEL
LIN {X 0,Y 563.5,Z 806.279,A -85,B 0,C 180,E1 2807.191,E2 2807.191} C_VEL
LIN {X 0,Y 564.28,Z 780.999,A -85,B 0,C 180,E1 2810.62,E2 2810.62} C_VEL
LIN {X 0,Y 565.385,Z 750.407,A -85,B 0,C 180,E1 2813.787,E2 2813.787} C_VEL
LIN {X 0,Y 566.654,Z 716.933,A -85,B 0,C 180,E1 2816.418,E2 2816.418} C_VEL
LIN {X 0,Y 567.849,Z 682.138,A -85,B 0,C 180,E1 2818.455,E2 2818.455} C_VEL
LIN {X 0,Y 568.884,Z 646.471,A -85,B 0,C 180,E1 2819.932,E2 2819.932} C_VEL
LIN {X 0,Y 569.583,Z 608.13,A -85,B 0,C 180,E1 2820.922,E2 2820.922} C_VEL
LIN {X 0,Y 568.82,Z 572.556,A -85,B 0,C 180,E1 2821.512,E2 2821.512} C_VEL
LIN {X 0,Y 562.295,Z 557.03,A -85,B 0,C 180,E1 2822.193,E2 2822.193} C_VEL
LIN {X 0,Y 561.931,Z 557.03,A -85,B 0,C 180,E1 2828.619,E2 2828.619} C_VEL
LIN {X 0,Y 562.014,Z 557.03,A -85,B 0,C 180,E1 2834.462,E2 2834.462} C_VEL
LIN {X 0,Y 562.069,Z 557.03,A -85,B 0,C 180,E1 2839.726,E2 2839.726} C_VEL
LIN {X 0,Y 561.991,Z 557.03,A -85,B 0,C 180,E1 2845.548,E2 2845.548} C_VEL
LIN {X 0,Y 562.05,Z 557.03,A -85,B 0,C 180,E1 2850.997,E2 2850.997} C_VEL
LIN {X 0,Y 562.171,Z 557.03,A -85,B 0,C 180,E1 2856.305,E2 2856.305} C_VEL
LIN {X 0,Y 562.29,Z 557.03,A -85,B 0,C 180,E1 2861.149,E2 2861.149} C_VEL
LIN {X 0,Y 561.935,Z 557.03,A -85,B 0,C 180,E1 2865.967,E2 2865.967} C_VEL
LIN {X 0,Y 562.257,Z 557.03,A -85,B 0,C 180,E1 2870.702,E2 2870.702} C_VEL
LIN {X 0,Y 562.332,Z 557.03,A -85,B 0,C 180,E1 2875.367,E2 2875.367} C_VEL
LIN {X 0,Y 562.392,Z 557.03,A -85,B 0,C 180,E1 2880,E2 2880} C_VEL
LIN {X 0,Y 562.358,Z 557.03,A -85,B 0,C 180,E1 2885.019,E2 2885.019} C_VEL
LIN {X 0,Y 562.229,Z 557.03,A -85,B 0,C 180,E1 2890.865,E2 2890.865} C_VEL
LIN {X 0,Y 562.186,Z 557.03,A -85,B 0,C 180,E1 2895.622,E2 2895.622} C_VEL
LIN {X 0,Y 562.224,Z 557.03,A -85,B 0,C 180,E1 2900.491,E2 2900.491} C_VEL
LIN {X 0,Y 562.107,Z 557.03,A -85,B 0,C 180,E1 2905.527,E2 2905.527} C_VEL
LIN {X 0,Y 562.035,Z 557.03,A -85,B 0,C 180,E1 2910.783,E2 2910.783} C_VEL
LIN {X 0,Y 562,Z 557.03,A -85,B 0,C 180,E1 2916.345,E2 2916.345} C_VEL
LIN {X 0,Y 561.926,Z 557.03,A -85,B 0,C 180,E1 2922.341,E2 2922.341} C_VEL
LIN {X 0,Y 562.06,Z 557.03,A -85,B 0,C 180,E1 2927.667,E2 2927.667} C_VEL
LIN {X 0,Y 562.115,Z 557.03,A -85,B 0,C 180,E1 2933.899,E2 2933.899} C_VEL
LIN {X 0,Y 562.1,Z 557.03,A -85,B 0,C 180,E1 2939.528,E2 2939.528} C_VEL
LIN {X 0,Y 562.132,Z 557.629,A -85,B 0,C 180,E1 2942.476,E2 2942.476} C_VEL
LIN {X 0,Y 567.989,Z 574.608,A -85,B 0,C 180,E1 2943.019,E2 2943.019} C_VEL
LIN {X 0,Y 567.47,Z 615.35,A -85,B 0,C 180,E1 2943.834,E2 2943.834} C_VEL
LIN {X 0,Y 566.703,Z 651.543,A -85,B 0,C 180,E1 2945.206,E2 2945.206} C_VEL
LIN {X 0,Y 565.74,Z 684.55,A -85,B 0,C 180,E1 2947.065,E2 2947.065} C_VEL
LIN {X 0,Y 564.752,Z 715.893,A -85,B 0,C 180,E1 2949.5,E2 2949.5} C_VEL
LIN {X 0,Y 563.834,Z 743.463,A -85,B 0,C 180,E1 2952.378,E2 2952.378} C_VEL
LIN {X 0,Y 563.222,Z 767.035,A -85,B 0,C 180,E1 2955.692,E2 2955.692} C_VEL
LIN {X 0,Y 562.838,Z 784.922,A -85,B 0,C 180,E1 2959.146,E2 2959.146} C_VEL
LIN {X 0,Y 562.692,Z 797.384,A -85,B 0,C 180,E1 2962.657,E2 2962.657} C_VEL
LIN {X 0,Y 562.649,Z 804.738,A -85,B 0,C 180,E1 2966.142,E2 2966.142} C_VEL
LIN {X 0,Y 562.584,Z 807.496,A -85,B 0,C 180,E1 2970,E2 2970} C_VEL
LIN {X 0,Y 562.686,Z 804.601,A -85,B 0,C 180,E1 2973.857,E2 2973.857} C_VEL
LIN {X 0,Y 562.791,Z 795.974,A -85,B 0,C 180,E1 2977.73,E2 2977.73} C_VEL
LIN {X 0,Y 562.999,Z 781.447,A -85,B 0,C 180,E1 2981.542,E2 2981.542} C_VEL
LIN {X 0,Y 563.411,Z 761.792,A -85,B 0,C 180,E1 2985.047,E2 2985.047} C_VEL
LIN {X 0,Y 564.054,Z 736.928,A -85,B 0,C 180,E1 2988.29,E2 2988.29} C_VEL
LIN {X 0,Y 564.99,Z 707.908,A -85,B 0,C 180,E1 2991.106,E2 2991.106} C_VEL
LIN {X 0,Y 566.025,Z 675.65,A -85,B 0,C 180,E1 2993.41,E2 2993.41} C_VEL
LIN {X 0,Y 566.941,Z 640.443,A -85,B 0,C 180,E1 2995.194,E2 2995.194} C_VEL
LIN {X 0,Y 567.69,Z 603.304,A -85,B 0,C 180,E1 2996.391,E2 2996.391} C_VEL
LIN {X 0,Y 567.151,Z 569.778,A -85,B 0,C 180,E1 2997.001,E2 2997.001} C_VEL
LIN {X 0,Y 562.394,Z 557.03,A -85,B 0,C 180,E1 2997.488,E2 2997.488} C_VEL
LIN {X 0,Y 562.095,Z 557.03,A -85,B 0,C 180,E1 3003.39,E2 3003.39} C_VEL
LIN {X 0,Y 561.965,Z 557.03,A -85,B 0,C 180,E1 3008.624,E2 3008.624} C_VEL
LIN {X 0,Y 562.012,Z 557.03,A -85,B 0,C 180,E1 3014.462,E2 3014.462} C_VEL
LIN {X 0,Y 562.041,Z 557.03,A -85,B 0,C 180,E1 3019.724,E2 3019.724} C_VEL
LIN {X 0,Y 561.984,Z 557.03,A -85,B 0,C 180,E1 3025.548,E2 3025.548} C_VEL
LIN {X 0,Y 562.047,Z 557.03,A -85,B 0,C 180,E1 3030.998,E2 3030.998} C_VEL
LIN {X 0,Y 562.212,Z 557.03,A -85,B 0,C 180,E1 3036.294,E2 3036.294} C_VEL
LIN {X 0,Y 562.295,Z 557.03,A -85,B 0,C 180,E1 3041.15,E2 3041.15} C_VEL
LIN {X 0,Y 562.45,Z 557.03,A -85,B 0,C 180,E1 3045.981,E2 3045.981} C_VEL
LIN {X 0,Y 562.376,Z 557.03,A -85,B 0,C 180,E1 3052.265,E2 3052.265} C_VEL
LIN {X 0,Y 562.504,Z 557.03,A -85,B 0,C 180,E1 3056.915,E2 3056.915} C_VEL
LIN {X 0,Y 562.593,Z 557.03,A -85,B 0,C 180,E1 3061.542,E2 3061.542} C_VEL
LIN {X 0,Y 562.248,Z 557.03,A -85,B 0,C 180,E1 3067.738,E2 3067.738} C_VEL
LIN {X 0,Y 562.221,Z 557.03,A -85,B 0,C 180,E1 3072.441,E2 3072.441} C_VEL
LIN {X 0,Y 562.174,Z 557.03,A -85,B 0,C 180,E1 3074.469,E2 3074.469} C_VEL
LIN {X 0,Y 558.185,Z 557.03,A -85,B 0,C 180,E1 3076.211,E2 3076.211} C_VEL
LIN {X 0,Y 554.188,Z 557.03,A -85,B 0,C 180,E1 3077.978,E2 3077.978} C_VEL
LIN {X 0,Y 554.241,Z 557.03,A -85,B 0,C 180,E1 3082.484,E2 3082.484} C_VEL
LIN {X 0,Y 554.15,Z 557.03,A -85,B 0,C 180,E1 3087.674,E2 3087.674} C_VEL
LIN {X 0,Y 554.068,Z 557.03,A -85,B 0,C 180,E1 3093.126,E2 3093.126} C_VEL
LIN {X 0,Y 554.151,Z 557.03,A -85,B 0,C 180,E1 3098.93,E2 3098.93} C_VEL
LIN {X 0,Y 554.154,Z 557.03,A -85,B 0,C 180,E1 3104.736,E2 3104.736} C_VEL
LIN {X 0,Y 554.047,Z 557.03,A -85,B 0,C 180,E1 3111.059,E2 3111.059} C_VEL
LIN {X 0,Y 554.337,Z 557.077,A -85,B 0,C 180,E1 3117.333,E2 3117.333} C_VEL
LIN {X 0,Y 562.903,Z 578.358,A -85,B 0,C 180,E1 3118.204,E2 3118.204} C_VEL
LIN {X 0,Y 562.434,Z 625.796,A -85,B 0,C 180,E1 3119.045,E2 3119.045} C_VEL
LIN {X 0,Y 561.386,Z 664.311,A -85,B 0,C 180,E1 3120.33,E2 3120.33} C_VEL
LIN {X 0,Y 560.064,Z 702.333,A -85,B 0,C 180,E1 3122.27,E2 3122.27} C_VEL
LIN {X 0,Y 558.56,Z 737.142,A -85,B 0,C 180,E1 3124.729,E2 3124.729} C_VEL
LIN {X 0,Y 557.128,Z 768.238,A -85,B 0,C 180,E1 3127.638,E2 3127.638} C_VEL
LIN {X 0,Y 556.095,Z 795.24,A -85,B 0,C 180,E1 3130.931,E2 3130.931} C_VEL
LIN {X 0,Y 555.378,Z 817.274,A -85,B 0,C 180,E1 3134.438,E2 3134.438} C_VEL
LIN {X 0,Y 554.913,Z 834.828,A -85,B 0,C 180,E1 3138.192,E2 3138.192} C_VEL
LIN {X 0,Y 554.784,Z 847.614,A -85,B 0,C 180,E1 3142.158,E2 3142.158} C_VEL
LIN {X 0,Y 554.688,Z 853.933,A -85,B 0,C 180,E1 3145.303,E2 3145.303} C_VEL
LIN {X 0,Y 554.681,Z 857.084,A -85,B 0,C 180,E1 3148.436,E2 3148.436} C_VEL
LIN {X 0,Y 554.775,Z 857.084,A -85,B 0,C 180,E1 3151.564,E2 3151.564} C_VEL
LIN {X 0,Y 554.84,Z 852.534,A -85,B 0,C 180,E1 3155.583,E2 3155.583} C_VEL
LIN {X 0,Y 554.857,Z 842.104,A -85,B 0,C 180,E1 3159.777,E2 3159.777} C_VEL
LIN {X 0,Y 555.188,Z 826.216,A -85,B 0,C 180,E1 3163.805,E2 3163.805} C_VEL
LIN {X 0,Y 555.742,Z 805.575,A -85,B 0,C 180,E1 3167.547,E2 3167.547} C_VEL
LIN {X 0,Y 556.76,Z 779.246,A -85,B 0,C 180,E1 3171.12,E2 3171.12} C_VEL
LIN {X 0,Y 557.967,Z 749.797,A -85,B 0,C 180,E1 3174.18,E2 3174.18} C_VEL
LIN {X 0,Y 559.426,Z 716.229,A -85,B 0,C 180,E1 3176.837,E2 3176.837} C_VEL
LIN {X 0,Y 560.908,Z 680.661,A -85,B 0,C 180,E1 3178.916,E2 3178.916} C_VEL
LIN {X 0,Y 562.062,Z 645.235,A -85,B 0,C 180,E1 3180.376,E2 3180.376} C_VEL
LIN {X 0,Y 562.837,Z 607.614,A -85,B 0,C 180,E1 3181.343,E2 3181.343} C_VEL
LIN {X 0,Y 562.243,Z 575.225,A -85,B 0,C 180,E1 3181.884,E2 3181.884} C_VEL
LIN {X 0,Y 554.341,Z 557.03,A -85,B 0,C 180,E1 3182.733,E2 3182.733} C_VEL
LIN {X 0,Y 554.008,Z 557.03,A -85,B 0,C 180,E1 3188.945,E2 3188.945} C_VEL
LIN {X 0,Y 554.157,Z 557.03,A -85,B 0,C 180,E1 3195.265,E2 3195.265} C_VEL
LIN {X 0,Y 554.153,Z 557.03,A -85,B 0,C 180,E1 3201.071,E2 3201.071} C_VEL
LIN {X 0,Y 554.071,Z 557.03,A -85,B 0,C 180,E1 3206.874,E2 3206.874} C_VEL
LIN {X 0,Y 554.152,Z 557.03,A -85,B 0,C 180,E1 3212.326,E2 3212.326} C_VEL
LIN {X 0,Y 554.248,Z 557.03,A -85,B 0,C 180,E1 3218.247,E2 3218.247} C_VEL
LIN {X 0,Y 554.422,Z 557.03,A -85,B 0,C 180,E1 3222.903,E2 3222.903} C_VEL
LIN {X 0,Y 554.354,Z 557.03,A -85,B 0,C 180,E1 3229.494,E2 3229.494} C_VEL
LIN {X 0,Y 554.455,Z 557.03,A -85,B 0,C 180,E1 3235.301,E2 3235.301} C_VEL
LIN {X 0,Y 554.492,Z 557.03,A -85,B 0,C 180,E1 3240,E2 3240} C_VEL
LIN {X 0,Y 554.518,Z 557.03,A -85,B 0,C 180,E1 3244.698,E2 3244.698} C_VEL
LIN {X 0,Y 554.337,Z 557.03,A -85,B 0,C 180,E1 3250.496,E2 3250.496} C_VEL
LIN {X 0,Y 554.276,Z 557.03,A -85,B 0,C 180,E1 3255.851,E2 3255.851} C_VEL
LIN {X 0,Y 554.285,Z 557.03,A -85,B 0,C 180,E1 3260.798,E2 3260.798} C_VEL
LIN {X 0,Y 554.157,Z 557.03,A -85,B 0,C 180,E1 3265.92,E2 3265.92} C_VEL
LIN {X 0,Y 554.09,Z 557.03,A -85,B 0,C 180,E1 3271.274,E2 3271.274} C_VEL
LIN {X 0,Y 554.013,Z 557.03,A -85,B 0,C 180,E1 3276.955,E2 3276.955} C_VEL
LIN {X 0,Y 554.05,Z 557.03,A -85,B 0,C 180,E1 3283.088,E2 3283.088} C_VEL
LIN {X 0,Y 554.142,Z 557.03,A -85,B 0,C 180,E1 3289.024,E2 3289.024} C_VEL
LIN {X 0,Y 554.087,Z 557.03,A -85,B 0,C 180,E1 3295.054,E2 3295.054} C_VEL
LIN {X 0,Y 554.147,Z 557.03,A -85,B 0,C 180,E1 3300.955,E2 3300.955} C_VEL
LIN {X 0,Y 554.162,Z 557.03,A -85,B 0,C 180,E1 3302.025,E2 3302.025} C_VEL
LIN {X 0,Y 560.955,Z 577.028,A -85,B 0,C 180,E1 3302.687,E2 3302.687} C_VEL
LIN {X 0,Y 560.328,Z 617.266,A -85,B 0,C 180,E1 3303.538,E2 3303.538} C_VEL
LIN {X 0,Y 559.427,Z 652.95,A -85,B 0,C 180,E1 3304.932,E2 3304.932} C_VEL
LIN {X 0,Y 558.315,Z 685.785,A -85,B 0,C 180,E1 3306.828,E2 3306.828} C_VEL
LIN {X 0,Y 557.095,Z 718.194,A -85,B 0,C 180,E1 3309.419,E2 3309.419} C_VEL
LIN {X 0,Y 556.071,Z 745.189,A -85,B 0,C 180,E1 3312.344,E2 3312.344} C_VEL
LIN {X 0,Y 555.418,Z 767.032,A -85,B 0,C 180,E1 3315.487,E2 3315.487} C_VEL
LIN {X 0,Y 554.991,Z 784.919,A -85,B 0,C 180,E1 3318.991,E2 3318.991} C_VEL
LIN {X 0,Y 554.831,Z 797.383,A -85,B 0,C 180,E1 3322.552,E2 3322.552} C_VEL
LIN {X 0,Y 554.775,Z 804.738,A -85,B 0,C 180,E1 3326.087,E2 3326.087} C_VEL
LIN {X 0,Y 554.698,Z 807.495,A -85,B 0,C 180,E1 3330,E2 3330} C_VEL
LIN {X 0,Y 554.815,Z 804.602,A -85,B 0,C 180,E1 3333.912,E2 3333.912} C_VEL
LIN {X 0,Y 554.91,Z 795.977,A -85,B 0,C 180,E1 3337.841,E2 3337.841} C_VEL
LIN {X 0,Y 555.115,Z 782.784,A -85,B 0,C 180,E1 3341.405,E2 3341.405} C_VEL
LIN {X 0,Y 555.611,Z 762.87,A -85,B 0,C 180,E1 3345.1,E2 3345.1} C_VEL
LIN {X 0,Y 556.332,Z 739.211,A -85,B 0,C 180,E1 3348.286,E2 3348.286} C_VEL
LIN {X 0,Y 557.386,Z 710.307,A -85,B 0,C 180,E1 3351.199,E2 3351.199} C_VEL
LIN {X 0,Y 558.619,Z 677.569,A -85,B 0,C 180,E1 3353.619,E2 3353.619} C_VEL
LIN {X 0,Y 559.621,Z 643.167,A -85,B 0,C 180,E1 3355.427,E2 3355.427} C_VEL
LIN {X 0,Y 560.549,Z 605.773,A -85,B 0,C 180,E1 3356.688,E2 3356.688} C_VEL
LIN {X 0,Y 560.169,Z 571.966,A -85,B 0,C 180,E1 3357.336,E2 3357.336} C_VEL
LIN {X 0,Y 554.401,Z 557.03,A -85,B 0,C 180,E1 3357.884,E2 3357.884} C_VEL
LIN {X 0,Y 554.186,Z 557.03,A -85,B 0,C 180,E1 3363.12,E2 3363.12} C_VEL
LIN {X 0,Y 554.042,Z 557.03,A -85,B 0,C 180,E1 3368.941,E2 3368.941} C_VEL
LIN {X 0,Y 554.151,Z 557.03,A -85,B 0,C 180,E1 3375.265,E2 3375.265} C_VEL
LIN {X 0,Y 554.127,Z 557.03,A -85,B 0,C 180,E1 3381.069,E2 3381.069} C_VEL
LIN {X 0,Y 554.048,Z 557.03,A -85,B 0,C 180,E1 3386.873,E2 3386.873} C_VEL
LIN {X 0,Y 554.178,Z 557.03,A -85,B 0,C 180,E1 3392.328,E2 3392.328} C_VEL
LIN {X 0,Y 554.28,Z 557.03,A -85,B 0,C 180,E1 3398.237,E2 3398.237} C_VEL
LIN {X 0,Y 554.399,Z 557.03,A -85,B 0,C 180,E1 3404.153,E2 3404.153} C_VEL
LIN {X 0,Y 554.374,Z 557.03,A -85,B 0,C 180,E1 3409.48,E2 3409.48} C_VEL
LIN {X 0,Y 554.521,Z 557.03,A -85,B 0,C 180,E1 3415.302,E2 3415.302} C_VEL
LIN {X 0,Y 554.682,Z 557.03,A -85,B 0,C 180,E1 3421.564,E2 3421.564} C_VEL
LIN {X 0,Y 554.335,Z 557.03,A -85,B 0,C 180,E1 3427.849,E2 3427.849} C_VEL
LIN {X 0,Y 554.298,Z 557.03,A -85,B 0,C 180,E1 3432.621,E2 3432.621} C_VEL
LIN {X 0,Y 554.188,Z 557.03,A -85,B 0,C 180,E1 3437.978,E2 3437.978} C_VEL
LIN {X 0,Y 550.285,Z 557.03,A -85,B 0,C 180,E1 3439.744,E2 3439.744} C_VEL
LIN {X 0,Y 546.313,Z 557.03,A -85,B 0,C 180,E1 3441.535,E2 3441.535} C_VEL
LIN {X 0,Y 546.27,Z 557.03,A -85,B 0,C 180,E1 3447.512,E2 3447.512} C_VEL
LIN {X 0,Y 546.112,Z 557.03,A -85,B 0,C 180,E1 3453.724,E2 3453.724} C_VEL
LIN {X 0,Y 546.224,Z 557.03,A -85,B 0,C 180,E1 3459.605,E2 3459.605} C_VEL
LIN {X 0,Y 546.205,Z 557.03,A -85,B 0,C 180,E1 3463.888,E2 3463.888} C_VEL
LIN {X 0,Y 546.13,Z 557.03,A -85,B 0,C 180,E1 3470.385,E2 3470.385} C_VEL
LIN {X 0,Y 546.398,Z 557.03,A -85,B 0,C 180,E1 3476.786,E2 3476.786} C_VEL
LIN {X 0,Y 556.228,Z 581.012,A -85,B 0,C 180,E1 3477.816,E2 3477.816} C_VEL
LIN {X 0,Y 555.629,Z 627.245,A -85,B 0,C 180,E1 3478.665,E2 3478.665} C_VEL
LIN {X 0,Y 554.424,Z 665.171,A -85,B 0,C 180,E1 3479.959,E2 3479.959} C_VEL
LIN {X 0,Y 552.954,Z 702.28,A -85,B 0,C 180,E1 3481.879,E2 3481.879} C_VEL
LIN {X 0,Y 551.255,Z 737.065,A -85,B 0,C 180,E1 3484.364,E2 3484.364} C_VEL
LIN {X 0,Y 549.618,Z 768.237,A -85,B 0,C 180,E1 3487.315,E2 3487.315} C_VEL
LIN {X 0,Y 548.398,Z 795.241,A -85,B 0,C 180,E1 3490.652,E2 3490.652} C_VEL
LIN {X 0,Y 547.573,Z 816.971,A -85,B 0,C 180,E1 3494.154,E2 3494.154} C_VEL
LIN {X 0,Y 547.043,Z 834.828,A -85,B 0,C 180,E1 3498.02,E2 3498.02} C_VEL
LIN {X 0,Y 546.955,Z 846.647,A -85,B 0,C 180,E1 3501.644,E2 3501.644} C_VEL
LIN {X 0,Y 546.797,Z 854.155,A -85,B 0,C 180,E1 3505.383,E2 3505.383} C_VEL
LIN {X 0,Y 546.78,Z 857.084,A -85,B 0,C 180,E1 3508.414,E2 3508.414} C_VEL
LIN {X 0,Y 546.87,Z 857.084,A -85,B 0,C 180,E1 3511.587,E2 3511.587} C_VEL
LIN {X 0,Y 546.944,Z 852.849,A -85,B 0,C 180,E1 3515.481,E2 3515.481} C_VEL
LIN {X 0,Y 547.003,Z 843.21,A -85,B 0,C 180,E1 3519.56,E2 3519.56} C_VEL
LIN {X 0,Y 547.352,Z 828.083,A -85,B 0,C 180,E1 3523.599,E2 3523.599} C_VEL
LIN {X 0,Y 547.964,Z 807.627,A -85,B 0,C 180,E1 3527.477,E2 3527.477} C_VEL
LIN {X 0,Y 549.118,Z 780.997,A -85,B 0,C 180,E1 3531.216,E2 3531.216} C_VEL
LIN {X 0,Y 550.47,Z 751.533,A -85,B 0,C 180,E1 3534.367,E2 3534.367} C_VEL
LIN {X 0,Y 552.157,Z 717.824,A -85,B 0,C 180,E1 3537.104,E2 3537.104} C_VEL
LIN {X 0,Y 553.802,Z 682.867,A -85,B 0,C 180,E1 3539.207,E2 3539.207} C_VEL
LIN {X 0,Y 555.18,Z 646.232,A -85,B 0,C 180,E1 3540.758,E2 3540.758} C_VEL
LIN {X 0,Y 556.083,Z 607.803,A -85,B 0,C 180,E1 3541.765,E2 3541.765} C_VEL
LIN {X 0,Y 555.487,Z 577.668,A -85,B 0,C 180,E1 3542.282,E2 3542.282} C_VEL
LIN {X 0,Y 546.366,Z 557.03,A -85,B 0,C 180,E1 3543.262,E2 3543.262} C_VEL
LIN {X 0,Y 546.092,Z 557.03,A -85,B 0,C 180,E1 3549.619,E2 3549.619} C_VEL
LIN {X 0,Y 546.209,Z 557.03,A -85,B 0,C 180,E1 3556.137,E2 3556.137} C_VEL
LIN {X 0,Y 546.217,Z 557.03,A -85,B 0,C 180,E1 3562.427,E2 3562.427} C_VEL
LIN {X 0,Y 546.18,Z 557.03,A -85,B 0,C 180,E1 3568.22,E2 3568.22} C_VEL
LIN {X 0,Y 546.268,Z 557.03,A -85,B 0,C 180,E1 3573.677,E2 3573.677} C_VEL
LIN {X 0,Y 546.4,Z 557.03,A -85,B 0,C 180,E1 3578.887,E2 3578.887} C_VEL
LIN {X 0,Y 546.383,Z 557.03,A -85,B 0,C 180,E1 3583.913,E2 3583.913} C_VEL
LIN {X 0,Y 546.445,Z 557.03,A -85,B 0,C 180,E1 3590.431,E2 3590.431} C_VEL
LIN {X 0,Y 546.582,Z 557.03,A -85,B 0,C 180,E1 3595.233,E2 3595.233} C_VEL
LIN {X 0,Y 546.591,Z 557.03,A -85,B 0,C 180,E1 3600,E2 3600} C_VEL
LIN {X 0,Y 546.609,Z 557.03,A -85,B 0,C 180,E1 3604.766,E2 3604.766} C_VEL
LIN {X 0,Y 546.514,Z 557.03,A -85,B 0,C 180,E1 3609.567,E2 3609.567} C_VEL
LIN {X 0,Y 546.479,Z 557.03,A -85,B 0,C 180,E1 3614.438,E2 3614.438} C_VEL
LIN {X 0,Y 546.415,Z 557.03,A -85,B 0,C 180,E1 3619.592,E2 3619.592} C_VEL
LIN {X 0,Y 546.309,Z 557.03,A -85,B 0,C 180,E1 3624.562,E2 3624.562} C_VEL
LIN {X 0,Y 546.155,Z 557.03,A -85,B 0,C 180,E1 3630.752,E2 3630.752} C_VEL
LIN {X 0,Y 546.082,Z 557.03,A -85,B 0,C 180,E1 3636.481,E2 3636.481} C_VEL
LIN {X 0,Y 546.109,Z 557.03,A -85,B 0,C 180,E1 3641.708,E2 3641.708} C_VEL
LIN {X 0,Y 546.201,Z 557.03,A -85,B 0,C 180,E1 3646.132,E2 3646.132} C_VEL
LIN {X 0,Y 546.211,Z 557.03,A -85,B 0,C 180,E1 3652.423,E2 3652.423} C_VEL
LIN {X 0,Y 546.17,Z 557.03,A -85,B 0,C 180,E1 3658.217,E2 3658.217} C_VEL
LIN {X 0,Y 546.25,Z 557.03,A -85,B 0,C 180,E1 3661.584,E2 3661.584} C_VEL
LIN {X 0,Y 553.951,Z 578.991,A -85,B 0,C 180,E1 3662.342,E2 3662.342} C_VEL
LIN {X 0,Y 553.197,Z 618.199,A -85,B 0,C 180,E1 3663.202,E2 3663.202} C_VEL
LIN {X 0,Y 552.172,Z 653.043,A -85,B 0,C 180,E1 3664.585,E2 3664.585} C_VEL
LIN {X 0,Y 550.942,Z 686.028,A -85,B 0,C 180,E1 3666.517,E2 3666.517} C_VEL
LIN {X 0,Y 549.591,Z 718.078,A -85,B 0,C 180,E1 3669.114,E2 3669.114} C_VEL
LIN {X 0,Y 548.399,Z 745.184,A -85,B 0,C 180,E1 3672.089,E2 3672.089} C_VEL
LIN {X 0,Y 547.604,Z 767.656,A -85,B 0,C 180,E1 3675.382,E2 3675.382} C_VEL
LIN {X 0,Y 547.121,Z 786.246,A -85,B 0,C 180,E1 3679.142,E2 3679.142} C_VEL
LIN {X 0,Y 546.968,Z 798.45,A -85,B 0,C 180,E1 3682.844,E2 3682.844} C_VEL
LIN {X 0,Y 546.856,Z 805.717,A -85,B 0,C 180,E1 3686.825,E2 3686.825} C_VEL
LIN {X 0,Y 546.799,Z 807.495,A -85,B 0,C 180,E1 3690,E2 3690} C_VEL
LIN {X 0,Y 546.915,Z 804.604,A -85,B 0,C 180,E1 3693.968,E2 3693.968} C_VEL
LIN {X 0,Y 547.055,Z 795.978,A -85,B 0,C 180,E1 3697.954,E2 3697.954} C_VEL
LIN {X 0,Y 547.247,Z 782.788,A -85,B 0,C 180,E1 3701.571,E2 3701.571} C_VEL
LIN {X 0,Y 547.828,Z 763.193,A -85,B 0,C 180,E1 3705.27,E2 3705.27} C_VEL
LIN {X 0,Y 548.673,Z 739.624,A -85,B 0,C 180,E1 3708.502,E2 3708.502} C_VEL
LIN {X 0,Y 549.815,Z 711.463,A -85,B 0,C 180,E1 3711.399,E2 3711.399} C_VEL
LIN {X 0,Y 551.251,Z 678.466,A -85,B 0,C 180,E1 3713.898,E2 3713.898} C_VEL
LIN {X 0,Y 552.424,Z 644.097,A -85,B 0,C 180,E1 3715.742,E2 3715.742} C_VEL
LIN {X 0,Y 553.434,Z 607.606,A -85,B 0,C 180,E1 3717.009,E2 3717.009} C_VEL
LIN {X 0,Y 553.262,Z 574.454,A -85,B 0,C 180,E1 3717.671,E2 3717.671} C_VEL
LIN {X 0,Y 546.445,Z 557.03,A -85,B 0,C 180,E1 3718.35,E2 3718.35} C_VEL
LIN {X 0,Y 546.191,Z 557.03,A -85,B 0,C 180,E1 3723.743,E2 3723.743} C_VEL
LIN {X 0,Y 546.125,Z 557.03,A -85,B 0,C 180,E1 3729.616,E2 3729.616} C_VEL
LIN {X 0,Y 546.201,Z 557.03,A -85,B 0,C 180,E1 3736.137,E2 3736.137} C_VEL
LIN {X 0,Y 546.198,Z 557.03,A -85,B 0,C 180,E1 3742.426,E2 3742.426} C_VEL
LIN {X 0,Y 546.147,Z 557.03,A -85,B 0,C 180,E1 3748.218,E2 3748.218} C_VEL
LIN {X 0,Y 546.329,Z 557.03,A -85,B 0,C 180,E1 3753.681,E2 3753.681} C_VEL
LIN {X 0,Y 546.429,Z 557.03,A -85,B 0,C 180,E1 3758.889,E2 3758.889} C_VEL
LIN {X 0,Y 546.501,Z 557.03,A -85,B 0,C 180,E1 3763.918,E2 3763.918} C_VEL
LIN {X 0,Y 546.467,Z 557.03,A -85,B 0,C 180,E1 3768.818,E2 3768.818} C_VEL
LIN {X 0,Y 546.491,Z 557.03,A -85,B 0,C 180,E1 3773.638,E2 3773.638} C_VEL
LIN {X 0,Y 546.522,Z 557.03,A -85,B 0,C 180,E1 3778.413,E2 3778.413} C_VEL
LIN {X 0,Y 546.501,Z 557.03,A -85,B 0,C 180,E1 3783.176,E2 3783.176} C_VEL
LIN {X 0,Y 546.423,Z 557.03,A -85,B 0,C 180,E1 3787.963,E2 3787.963} C_VEL
LIN {X 0,Y 546.378,Z 557.03,A -85,B 0,C 180,E1 3792.807,E2 3792.807} C_VEL
LIN {X 0,Y 546.28,Z 557.03,A -85,B 0,C 180,E1 3797.97,E2 3797.97} C_VEL
LIN {X 0,Y 546.313,Z 557.03,A -85,B 0,C 180,E1 3801.535,E2 3801.535} C_VEL
LIN {X 0,Y 542.325,Z 557.03,A -85,B 0,C 180,E1 3803.324,E2 3803.324} C_VEL
LIN {X 0,Y 538.37,Z 557.03,A -85,B 0,C 180,E1 3805.139,E2 3805.139} C_VEL
LIN {X 0,Y 538.275,Z 557.03,A -85,B 0,C 180,E1 3810.416,E2 3810.416} C_VEL
LIN {X 0,Y 538.235,Z 557.03,A -85,B 0,C 180,E1 3816.206,E2 3816.206} C_VEL
LIN {X 0,Y 538.233,Z 557.03,A -85,B 0,C 180,E1 3822.46,E2 3822.46} C_VEL
LIN {X 0,Y 538.147,Z 557.03,A -85,B 0,C 180,E1 3827.529,E2 3827.529} C_VEL
LIN {X 0,Y 538.205,Z 557.03,A -85,B 0,C 180,E1 3833.789,E2 3833.789} C_VEL
LIN {X 0,Y 538.437,Z 557.625,A -85,B 0,C 180,E1 3836.25,E2 3836.25} C_VEL
LIN {X 0,Y 549.524,Z 581.769,A -85,B 0,C 180,E1 3837.386,E2 3837.386} C_VEL
LIN {X 0,Y 548.845,Z 627.244,A -85,B 0,C 180,E1 3838.233,E2 3838.233} C_VEL
LIN {X 0,Y 547.565,Z 664.43,A -85,B 0,C 180,E1 3839.508,E2 3839.508} C_VEL
LIN {X 0,Y 545.952,Z 700.664,A -85,B 0,C 180,E1 3841.378,E2 3841.378} C_VEL
LIN {X 0,Y 544.03,Z 735.509,A -85,B 0,C 180,E1 3843.862,E2 3843.862} C_VEL
LIN {X 0,Y 542.273,Z 766.318,A -85,B 0,C 180,E1 3846.773,E2 3846.773} C_VEL
LIN {X 0,Y 540.797,Z 793.877,A -85,B 0,C 180,E1 3850.172,E2 3850.172} C_VEL
LIN {X 0,Y 539.774,Z 816.978,A -85,B 0,C 180,E1 3853.92,E2 3853.92} C_VEL
LIN {X 0,Y 539.188,Z 834.829,A -85,B 0,C 180,E1 3857.843,E2 3857.843} C_VEL
LIN {X 0,Y 539.054,Z 846.647,A -85,B 0,C 180,E1 3861.521,E2 3861.521} C_VEL
LIN {X 0,Y 538.916,Z 853.933,A -85,B 0,C 180,E1 3865.165,E2 3865.165} C_VEL
LIN {X 0,Y 538.896,Z 857.084,A -85,B 0,C 180,E1 3868.39,E2 3868.39} C_VEL
LIN {X 0,Y 538.979,Z 857.084,A -85,B 0,C 180,E1 3871.61,E2 3871.61} C_VEL
LIN {X 0,Y 539.02,Z 852.725,A -85,B 0,C 180,E1 3875.642,E2 3875.642} C_VEL
LIN {X 0,Y 539.098,Z 843.211,A -85,B 0,C 180,E1 3879.701,E2 3879.701} C_VEL
LIN {X 0,Y 539.5,Z 828.13,A -85,B 0,C 180,E1 3883.79,E2 3883.79} C_VEL
LIN {X 0,Y 540.208,Z 808.054,A -85,B 0,C 180,E1 3887.662,E2 3887.662} C_VEL
LIN {X 0,Y 541.533,Z 781.181,A -85,B 0,C 180,E1 3891.506,E2 3891.506} C_VEL
LIN {X 0,Y 543.099,Z 751.535,A -85,B 0,C 180,E1 3894.719,E2 3894.719} C_VEL
LIN {X 0,Y 544.992,Z 717.842,A -85,B 0,C 180,E1 3897.489,E2 3897.489} C_VEL
LIN {X 0,Y 546.806,Z 683.016,A -85,B 0,C 180,E1 3899.61,E2 3899.61} C_VEL
LIN {X 0,Y 548.34,Z 646.018,A -85,B 0,C 180,E1 3901.192,E2 3901.192} C_VEL
LIN {X 0,Y 549.381,Z 607.803,A -85,B 0,C 180,E1 3902.199,E2 3902.199} C_VEL
LIN {X 0,Y 549.125,Z 580.936,A -85,B 0,C 180,E1 3902.653,E2 3902.653} C_VEL
LIN {X 0,Y 538.378,Z 557.03,A -85,B 0,C 180,E1 3903.855,E2 3903.855} C_VEL
LIN {X 0,Y 538.129,Z 557.03,A -85,B 0,C 180,E1 3910.325,E2 3910.325} C_VEL
LIN {X 0,Y 538.216,Z 557.03,A -85,B 0,C 180,E1 3915.313,E2 3915.313} C_VEL
LIN {X 0,Y 538.304,Z 557.03,A -85,B 0,C 180,E1 3921.776,E2 3921.776} C_VEL
LIN {X 0,Y 538.203,Z 557.03,A -85,B 0,C 180,E1 3927.692,E2 3927.692} C_VEL
LIN {X 0,Y 538.36,Z 557.03,A -85,B 0,C 180,E1 3933.26,E2 3933.26} C_VEL
LIN {X 0,Y 538.442,Z 557.03,A -85,B 0,C 180,E1 3938.56,E2 3938.56} C_VEL
LIN {X 0,Y 538.468,Z 557.03,A -85,B 0,C 180,E1 3943.67,E2 3943.67} C_VEL
LIN {X 0,Y 538.525,Z 557.03,A -85,B 0,C 180,E1 3950.289,E2 3950.289} C_VEL
LIN {X 0,Y 538.678,Z 557.03,A -85,B 0,C 180,E1 3955.163,E2 3955.163} C_VEL
LIN {X 0,Y 538.709,Z 557.03,A -85,B 0,C 180,E1 3960,E2 3960} C_VEL
LIN {X 0,Y 538.695,Z 557.03,A -85,B 0,C 180,E1 3964.836,E2 3964.836} C_VEL
LIN {X 0,Y 538.535,Z 557.03,A -85,B 0,C 180,E1 3970.262,E2 3970.262} C_VEL
LIN {X 0,Y 538.543,Z 557.03,A -85,B 0,C 180,E1 3974.655,E2 3974.655} C_VEL
LIN {X 0,Y 538.51,Z 557.03,A -85,B 0,C 180,E1 3979.716,E2 3979.716} C_VEL
LIN {X 0,Y 538.305,Z 557.03,A -85,B 0,C 180,E1 3985.836,E2 3985.836} C_VEL
LIN {X 0,Y 538.269,Z 557.03,A -85,B 0,C 180,E1 3990.415,E2 3990.415} C_VEL
LIN {X 0,Y 538.174,Z 557.03,A -85,B 0,C 180,E1 3996.21,E2 3996.21} C_VEL
LIN {X 0,Y 538.132,Z 557.03,A -85,B 0,C 180,E1 4002.469,E2 4002.469} C_VEL
LIN {X 0,Y 538.228,Z 557.03,A -85,B 0,C 180,E1 4007.536,E2 4007.536} C_VEL
LIN {X 0,Y 538.229,Z 557.03,A -85,B 0,C 180,E1 4013.79,E2 4013.79} C_VEL
LIN {X 0,Y 538.261,Z 557.03,A -85,B 0,C 180,E1 4019.581,E2 4019.581} C_VEL
LIN {X 0,Y 538.342,Z 557.03,A -85,B 0,C 180,E1 4021.141,E2 4021.141} C_VEL
LIN {X 0,Y 546.967,Z 580.931,A -85,B 0,C 180,E1 4021.987,E2 4021.987} C_VEL
LIN {X 0,Y 546.092,Z 619.432,A -85,B 0,C 180,E1 4022.868,E2 4022.868} C_VEL
LIN {X 0,Y 544.906,Z 654.77,A -85,B 0,C 180,E1 4024.312,E2 4024.312} C_VEL
LIN {X 0,Y 543.458,Z 688.744,A -85,B 0,C 180,E1 4026.369,E2 4026.369} C_VEL
LIN {X 0,Y 541.89,Z 720.698,A -85,B 0,C 180,E1 4029.07,E2 4029.07} C_VEL
LIN {X 0,Y 540.572,Z 748.18,A -85,B 0,C 180,E1 4032.215,E2 4032.215} C_VEL
LIN {X 0,Y 539.752,Z 771.177,A -85,B 0,C 180,E1 4035.792,E2 4035.792} C_VEL
LIN {X 0,Y 539.234,Z 787.492,A -85,B 0,C 180,E1 4039.311,E2 4039.311} C_VEL
LIN {X 0,Y 539.072,Z 798.448,A -85,B 0,C 180,E1 4042.739,E2 4042.739} C_VEL
LIN {X 0,Y 538.971,Z 805.716,A -85,B 0,C 180,E1 4046.779,E2 4046.779} C_VEL
LIN {X 0,Y 538.907,Z 807.495,A -85,B 0,C 180,E1 4050,E2 4050} C_VEL
LIN {X 0,Y 538.994,Z 804.85,A -85,B 0,C 180,E1 4053.862,E2 4053.862} C_VEL
LIN {X 0,Y 539.154,Z 797.127,A -85,B 0,C 180,E1 4057.665,E2 4057.665} C_VEL
LIN {X 0,Y 539.355,Z 784.532,A -85,B 0,C 180,E1 4061.332,E2 4061.332} C_VEL
LIN {X 0,Y 539.908,Z 766.883,A -85,B 0,C 180,E1 4064.874,E2 4064.874} C_VEL
LIN {X 0,Y 540.871,Z 743.08,A -85,B 0,C 180,E1 4068.356,E2 4068.356} C_VEL
LIN {X 0,Y 542.198,Z 714.922,A -85,B 0,C 180,E1 4071.393,E2 4071.393} C_VEL
LIN {X 0,Y 543.667,Z 683.225,A -85,B 0,C 180,E1 4073.924,E2 4073.924} C_VEL
LIN {X 0,Y 545.132,Z 647.48,A -85,B 0,C 180,E1 4075.958,E2 4075.958} C_VEL
LIN {X 0,Y 546.356,Z 610.365,A -85,B 0,C 180,E1 4077.31,E2 4077.31} C_VEL
LIN {X 0,Y 546.314,Z 576.587,A -85,B 0,C 180,E1 4078.023,E2 4078.023} C_VEL
LIN {X 0,Y 538.515,Z 557.03,A -85,B 0,C 180,E1 4078.782,E2 4078.782} C_VEL
LIN {X 0,Y 538.175,Z 557.03,A -85,B 0,C 180,E1 4085.334,E2 4085.334} C_VEL
LIN {X 0,Y 538.145,Z 557.03,A -85,B 0,C 180,E1 4090.573,E2 4090.573} C_VEL
LIN {X 0,Y 538.241,Z 557.03,A -85,B 0,C 180,E1 4097.001,E2 4097.001} C_VEL
LIN {X 0,Y 538.265,Z 557.03,A -85,B 0,C 180,E1 4101.961,E2 4101.961} C_VEL
LIN {X 0,Y 538.178,Z 557.03,A -85,B 0,C 180,E1 4107.691,E2 4107.691} C_VEL
LIN {X 0,Y 538.394,Z 557.03,A -85,B 0,C 180,E1 4113.262,E2 4113.262} C_VEL
LIN {X 0,Y 538.472,Z 557.03,A -85,B 0,C 180,E1 4118.562,E2 4118.562} C_VEL
LIN {X 0,Y 538.564,Z 557.03,A -85,B 0,C 180,E1 4123.674,E2 4123.674} C_VEL
LIN {X 0,Y 538.567,Z 557.03,A -85,B 0,C 180,E1 4128.652,E2 4128.652} C_VEL
LIN {X 0,Y 538.583,Z 557.03,A -85,B 0,C 180,E1 4133.544,E2 4133.544} C_VEL
LIN {X 0,Y 538.652,Z 557.03,A -85,B 0,C 180,E1 4138.39,E2 4138.39} C_VEL
LIN {X 0,Y 538.606,Z 557.03,A -85,B 0,C 180,E1 4143.223,E2 4143.223} C_VEL
LIN {X 0,Y 538.511,Z 557.03,A -85,B 0,C 180,E1 4148.081,E2 4148.081} C_VEL
LIN {X 0,Y 538.481,Z 557.03,A -85,B 0,C 180,E1 4152.998,E2 4152.998} C_VEL
LIN {X 0,Y 538.406,Z 557.03,A -85,B 0,C 180,E1 4158.018,E2 4158.018} C_VEL
LIN {X 0,Y 538.393,Z 557.03,A -85,B 0,C 180,E1 4163.184,E2 4163.184} C_VEL
LIN {X 0,Y 538.37,Z 557.03,A -85,B 0,C 180,E1 4165.139,E2 4165.139} C_VEL
LIN {X 0,Y 537.056,Z 557.03,A -85,B 0,C 180,E1 4166.061,E2 4166.061} C_VEL
LIN {X 0,Y 530.412,Z 557.03,A -85,B 0,C 180,E1 4168.572,E2 4168.572} C_VEL
LIN {X 0,Y 530.334,Z 557.03,A -85,B 0,C 180,E1 4168.81,E2 4168.81} C_VEL
LIN {X 0,Y 530.284,Z 557.03,A -85,B 0,C 180,E1 4174.82,E2 4174.82} C_VEL
LIN {X 0,Y 530.321,Z 557.03,A -85,B 0,C 180,E1 4181.041,E2 4181.041} C_VEL
LIN {X 0,Y 530.283,Z 557.03,A -85,B 0,C 180,E1 4186.746,E2 4186.746} C_VEL
LIN {X 0,Y 530.242,Z 557.03,A -85,B 0,C 180,E1 4193.157,E2 4193.157} C_VEL
LIN {X 0,Y 530.451,Z 557.644,A -85,B 0,C 180,E1 4195.672,E2 4195.672} C_VEL
LIN {X 0,Y 542.845,Z 584.292,A -85,B 0,C 180,E1 4196.973,E2 4196.973} C_VEL
LIN {X 0,Y 542.069,Z 628.675,A -85,B 0,C 180,E1 4197.831,E2 4197.831} C_VEL
LIN {X 0,Y 540.534,Z 667.299,A -85,B 0,C 180,E1 4199.206,E2 4199.206} C_VEL
LIN {X 0,Y 538.777,Z 702.565,A -85,B 0,C 180,E1 4201.09,E2 4201.09} C_VEL
LIN {X 0,Y 536.667,Z 736.992,A -85,B 0,C 180,E1 4203.608,E2 4203.608} C_VEL
LIN {X 0,Y 534.688,Z 768.236,A -85,B 0,C 180,E1 4206.645,E2 4206.645} C_VEL
LIN {X 0,Y 533.074,Z 795.243,A -85,B 0,C 180,E1 4210.073,E2 4210.073} C_VEL
LIN {X 0,Y 531.951,Z 818.073,A -85,B 0,C 180,E1 4213.889,E2 4213.889} C_VEL
LIN {X 0,Y 531.352,Z 834.829,A -85,B 0,C 180,E1 4217.661,E2 4217.661} C_VEL
LIN {X 0,Y 531.169,Z 846.647,A -85,B 0,C 180,E1 4221.394,E2 4221.394} C_VEL
LIN {X 0,Y 531.028,Z 853.933,A -85,B 0,C 180,E1 4225.094,E2 4225.094} C_VEL
LIN {X 0,Y 530.994,Z 857.084,A -85,B 0,C 180,E1 4228.366,E2 4228.366} C_VEL
LIN {X 0,Y 531.073,Z 857.084,A -85,B 0,C 180,E1 4231.634,E2 4231.634} C_VEL
LIN {X 0,Y 531.113,Z 852.725,A -85,B 0,C 180,E1 4235.727,E2 4235.727} C_VEL
LIN {X 0,Y 531.224,Z 843.211,A -85,B 0,C 180,E1 4239.847,E2 4239.847} C_VEL
LIN {X 0,Y 531.653,Z 827.326,A -85,B 0,C 180,E1 4244.188,E2 4244.188} C_VEL
LIN {X 0,Y 532.553,Z 806.273,A -85,B 0,C 180,E1 4248.224,E2 4248.224} C_VEL
LIN {X 0,Y 533.994,Z 779.944,A -85,B 0,C 180,E1 4251.979,E2 4251.979} C_VEL
LIN {X 0,Y 535.81,Z 750.182,A -85,B 0,C 180,E1 4255.211,E2 4255.211} C_VEL
LIN {X 0,Y 537.871,Z 716.689,A -85,B 0,C 180,E1 4257.969,E2 4257.969} C_VEL
LIN {X 0,Y 539.917,Z 681.785,A -85,B 0,C 180,E1 4260.093,E2 4260.093} C_VEL
LIN {X 0,Y 541.556,Z 645.772,A -85,B 0,C 180,E1 4261.637,E2 4261.637} C_VEL
LIN {X 0,Y 542.696,Z 608.544,A -85,B 0,C 180,E1 4262.631,E2 4262.631} C_VEL
LIN {X 0,Y 542.163,Z 582.655,A -85,B 0,C 180,E1 4263.099,E2 4263.099} C_VEL
LIN {X 0,Y 530.412,Z 557.03,A -85,B 0,C 180,E1 4264.388,E2 4264.388} C_VEL
LIN {X 0,Y 530.182,Z 557.03,A -85,B 0,C 180,E1 4271.058,E2 4271.058} C_VEL
LIN {X 0,Y 530.343,Z 557.03,A -85,B 0,C 180,E1 4276.755,E2 4276.755} C_VEL
LIN {X 0,Y 530.295,Z 557.03,A -85,B 0,C 180,E1 4283.076,E2 4283.076} C_VEL
LIN {X 0,Y 530.301,Z 557.03,A -85,B 0,C 180,E1 4289.077,E2 4289.077} C_VEL
LIN {X 0,Y 530.463,Z 557.03,A -85,B 0,C 180,E1 4294.653,E2 4294.653} C_VEL
LIN {X 0,Y 530.64,Z 557.03,A -85,B 0,C 180,E1 4300.318,E2 4300.318} C_VEL
LIN {X 0,Y 530.342,Z 557.03,A -85,B 0,C 180,E1 4306.086,E2 4306.086} C_VEL
LIN {X 0,Y 530.62,Z 557.03,A -85,B 0,C 180,E1 4311.798,E2 4311.798} C_VEL
LIN {X 0,Y 530.732,Z 557.03,A -85,B 0,C 180,E1 4316.831,E2 4316.831} C_VEL
LIN {X 0,Y 530.757,Z 557.03,A -85,B 0,C 180,E1 4321.634,E2 4321.634} C_VEL
LIN {X 0,Y 530.693,Z 557.03,A -85,B 0,C 180,E1 4326.552,E2 4326.552} C_VEL
LIN {X 0,Y 530.611,Z 557.03,A -85,B 0,C 180,E1 4331.521,E2 4331.521} C_VEL
LIN {X 0,Y 530.577,Z 557.03,A -85,B 0,C 180,E1 4336.579,E2 4336.579} C_VEL
LIN {X 0,Y 530.537,Z 557.03,A -85,B 0,C 180,E1 4341.775,E2 4341.775} C_VEL
LIN {X 0,Y 530.329,Z 557.03,A -85,B 0,C 180,E1 4347.744,E2 4347.744} C_VEL
LIN {X 0,Y 530.324,Z 557.03,A -85,B 0,C 180,E1 4354.112,E2 4354.112} C_VEL
LIN {X 0,Y 530.178,Z 557.03,A -85,B 0,C 180,E1 4359.551,E2 4359.551} C_VEL
LIN {X 0,Y 530.294,Z 557.03,A -85,B 0,C 180,E1 4365.539,E2 4365.539} C_VEL
LIN {X 0,Y 530.299,Z 557.03,A -85,B 0,C 180,E1 4371.088,E2 4371.088} C_VEL
LIN {X 0,Y 530.265,Z 557.03,A -85,B 0,C 180,E1 4377.146,E2 4377.146} C_VEL
LIN {X 0,Y 530.407,Z 557.03,A -85,B 0,C 180,E1 4380.617,E2 4380.617} C_VEL
LIN {X 0,Y 539.987,Z 582.831,A -85,B 0,C 180,E1 4381.626,E2 4381.626} C_VEL
LIN {X 0,Y 539.027,Z 619.92,A -85,B 0,C 180,E1 4382.5,E2 4382.5} C_VEL
LIN {X 0,Y 537.683,Z 655.807,A -85,B 0,C 180,E1 4383.996,E2 4383.996} C_VEL
LIN {X 0,Y 536.004,Z 690.497,A -85,B 0,C 180,E1 4386.153,E2 4386.153} C_VEL
LIN {X 0,Y 534.337,Z 721.487,A -85,B 0,C 180,E1 4388.843,E2 4388.843} C_VEL
LIN {X 0,Y 532.915,Z 748.174,A -85,B 0,C 180,E1 4391.951,E2 4391.951} C_VEL
LIN {X 0,Y 531.955,Z 770.153,A -85,B 0,C 180,E1 4395.383,E2 4395.383} C_VEL
LIN {X 0,Y 531.372,Z 787.49,A -85,B 0,C 180,E1 4399.151,E2 4399.151} C_VEL
LIN {X 0,Y 531.195,Z 798.447,A -85,B 0,C 180,E1 4402.631,E2 4402.631} C_VEL
LIN {X 0,Y 531.069,Z 805.715,A -85,B 0,C 180,E1 4406.731,E2 4406.731} C_VEL
LIN {X 0,Y 531.007,Z 807.495,A -85,B 0,C 180,E1 4410,E2 4410} C_VEL
LIN {X 0,Y 531.096,Z 804.907,A -85,B 0,C 180,E1 4413.881,E2 4413.881} C_VEL
LIN {X 0,Y 531.29,Z 797.129,A -85,B 0,C 180,E1 4417.779,E2 4417.779} C_VEL
LIN {X 0,Y 531.5,Z 784.534,A -85,B 0,C 180,E1 4421.502,E2 4421.502} C_VEL
LIN {X 0,Y 532.213,Z 765.96,A -85,B 0,C 180,E1 4425.257,E2 4425.257} C_VEL
LIN {X 0,Y 533.284,Z 741.386,A -85,B 0,C 180,E1 4428.841,E2 4428.841} C_VEL
LIN {X 0,Y 534.703,Z 713.872,A -85,B 0,C 180,E1 4431.808,E2 4431.808} C_VEL
LIN {X 0,Y 536.452,Z 681.685,A -85,B 0,C 180,E1 4434.378,E2 4434.378} C_VEL
LIN {X 0,Y 538.083,Z 645.497,A -85,B 0,C 180,E1 4436.417,E2 4436.417} C_VEL
LIN {X 0,Y 539.325,Z 608.867,A -85,B 0,C 180,E1 4437.74,E2 4437.74} C_VEL
LIN {X 0,Y 539.354,Z 578.947,A -85,B 0,C 180,E1 4438.383,E2 4438.383} C_VEL
LIN {X 0,Y 530.502,Z 557.03,A -85,B 0,C 180,E1 4439.332,E2 4439.332} C_VEL
LIN {X 0,Y 530.293,Z 557.03,A -85,B 0,C 180,E1 4444.821,E2 4444.821} C_VEL
LIN {X 0,Y 530.198,Z 557.03,A -85,B 0,C 180,E1 4451.056,E2 4451.056} C_VEL
LIN {X 0,Y 530.335,Z 557.03,A -85,B 0,C 180,E1 4456.755,E2 4456.755} C_VEL
LIN {X 0,Y 530.272,Z 557.03,A -85,B 0,C 180,E1 4463.079,E2 4463.079} C_VEL
LIN {X 0,Y 530.279,Z 557.03,A -85,B 0,C 180,E1 4469.076,E2 4469.076} C_VEL
LIN {X 0,Y 530.52,Z 557.03,A -85,B 0,C 180,E1 4474.656,E2 4474.656} C_VEL
LIN {X 0,Y 530.66,Z 557.03,A -85,B 0,C 180,E1 4480.311,E2 4480.311} C_VEL
LIN {X 0,Y 530.721,Z 557.03,A -85,B 0,C 180,E1 4485.919,E2 4485.919} C_VEL
LIN {X 0,Y 530.739,Z 557.03,A -85,B 0,C 180,E1 4491.8,E2 4491.8} C_VEL
LIN {X 0,Y 530.889,Z 557.03,A -85,B 0,C 180,E1 4496.731,E2 4496.731} C_VEL
LIN {X 0,Y 530.971,Z 557.03,A -85,B 0,C 180,E1 4501.634,E2 4501.634} C_VEL
LIN {X 0,Y 530.842,Z 557.03,A -85,B 0,C 180,E1 4506.551,E2 4506.551} C_VEL
LIN {X 0,Y 530.661,Z 557.03,A -85,B 0,C 180,E1 4511.52,E2 4511.52} C_VEL
LIN {X 0,Y 530.526,Z 557.03,A -85,B 0,C 180,E1 4516.581,E2 4516.581} C_VEL
LIN {X 0,Y 530.518,Z 557.03,A -85,B 0,C 180,E1 4521.777,E2 4521.777} C_VEL
LIN {X 0,Y 530.353,Z 557.03,A -85,B 0,C 180,E1 4527.751,E2 4527.751} C_VEL
LIN {X 0,Y 530.334,Z 557.03,A -85,B 0,C 180,E1 4528.81,E2 4528.81} C_VEL
LIN {X 0,Y 527.807,Z 557.03,A -85,B 0,C 180,E1 4530.199,E2 4530.199} C_VEL
LIN {X 0,Y 522.421,Z 557.03,A -85,B 0,C 180,E1 4532.28,E2 4532.28} C_VEL
LIN {X 0,Y 522.344,Z 557.03,A -85,B 0,C 180,E1 4532.52,E2 4532.52} C_VEL
LIN {X 0,Y 522.359,Z 557.03,A -85,B 0,C 180,E1 4538.502,E2 4538.502} C_VEL
LIN {X 0,Y 522.417,Z 557.03,A -85,B 0,C 180,E1 4544.068,E2 4544.068} C_VEL
LIN {X 0,Y 522.298,Z 557.03,A -85,B 0,C 180,E1 4550.377,E2 4550.377} C_VEL
LIN {X 0,Y 522.431,Z 557.03,A -85,B 0,C 180,E1 4555.039,E2 4555.039} C_VEL
LIN {X 0,Y 536.27,Z 586.784,A -85,B 0,C 180,E1 4556.555,E2 4556.555} C_VEL
LIN {X 0,Y 535.368,Z 628.674,A -85,B 0,C 180,E1 4557.379,E2 4557.379} C_VEL
LIN {X 0,Y 533.745,Z 666.732,A -85,B 0,C 180,E1 4558.744,E2 4558.744} C_VEL
LIN {X 0,Y 531.648,Z 703.891,A -85,B 0,C 180,E1 4560.756,E2 4560.756} C_VEL
LIN {X 0,Y 529.32,Z 738.377,A -85,B 0,C 180,E1 4563.339,E2 4563.339} C_VEL
LIN {X 0,Y 527.109,Z 769.857,A -85,B 0,C 180,E1 4566.479,E2 4566.479} C_VEL
LIN {X 0,Y 525.368,Z 796.7,A -85,B 0,C 180,E1 4569.988,E2 4569.988} C_VEL
LIN {X 0,Y 524.123,Z 819.157,A -85,B 0,C 180,E1 4573.857,E2 4573.857} C_VEL
LIN {X 0,Y 523.457,Z 836.368,A -85,B 0,C 180,E1 4577.896,E2 4577.896} C_VEL
LIN {X 0,Y 523.25,Z 847.614,A -85,B 0,C 180,E1 4581.682,E2 4581.682} C_VEL
LIN {X 0,Y 523.127,Z 853.934,A -85,B 0,C 180,E1 4585.019,E2 4585.019} C_VEL
LIN {X 0,Y 523.111,Z 857.084,A -85,B 0,C 180,E1 4588.342,E2 4588.342} C_VEL
LIN {X 0,Y 523.184,Z 857.085,A -85,B 0,C 180,E1 4591.659,E2 4591.659} C_VEL
LIN {X 0,Y 523.221,Z 852.725,A -85,B 0,C 180,E1 4595.813,E2 4595.813} C_VEL
LIN {X 0,Y 523.342,Z 843.211,A -85,B 0,C 180,E1 4599.997,E2 4599.997} C_VEL
LIN {X 0,Y 523.818,Z 827.822,A -85,B 0,C 180,E1 4604.287,E2 4604.287} C_VEL
LIN {X 0,Y 524.849,Z 806.272,A -85,B 0,C 180,E1 4608.501,E2 4608.501} C_VEL
LIN {X 0,Y 526.403,Z 780.331,A -85,B 0,C 180,E1 4612.264,E2 4612.264} C_VEL
LIN {X 0,Y 528.436,Z 750.417,A -85,B 0,C 180,E1 4615.565,E2 4615.565} C_VEL
LIN {X 0,Y 530.719,Z 717.231,A -85,B 0,C 180,E1 4618.339,E2 4618.339} C_VEL
LIN {X 0,Y 532.988,Z 681.536,A -85,B 0,C 180,E1 4620.539,E2 4620.539} C_VEL
LIN {X 0,Y 534.801,Z 645.54,A -85,B 0,C 180,E1 4622.092,E2 4622.092} C_VEL
LIN {X 0,Y 536.065,Z 607.961,A -85,B 0,C 180,E1 4623.096,E2 4623.096} C_VEL
LIN {X 0,Y 535.653,Z 585.496,A -85,B 0,C 180,E1 4623.509,E2 4623.509} C_VEL
LIN {X 0,Y 522.415,Z 557.03,A -85,B 0,C 180,E1 4625.021,E2 4625.021} C_VEL
LIN {X 0,Y 522.294,Z 557.03,A -85,B 0,C 180,E1 4631.092,E2 4631.092} C_VEL
LIN {X 0,Y 522.436,Z 557.03,A -85,B 0,C 180,E1 4636.429,E2 4636.429} C_VEL
LIN {X 0,Y 522.351,Z 557.03,A -85,B 0,C 180,E1 4642.508,E2 4642.508} C_VEL
LIN {X 0,Y 522.357,Z 557.03,A -85,B 0,C 180,E1 4648.554,E2 4648.554} C_VEL
